KUKA KRL program: MyProgram_134().src

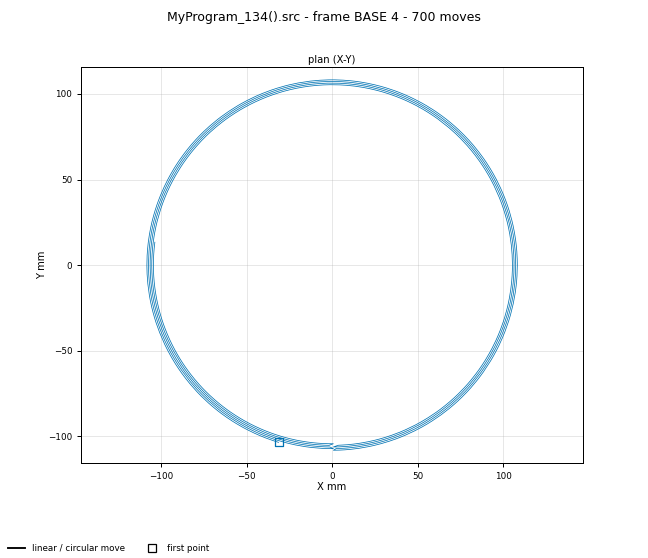
[picture p0: tool path of MyProgram_134().src in frame BASE 4, 700 of 700 moves have a stored position in this frame; points joined in program order, loops and branches not executed]
&ACCESS RVP
&REL 1
&PARAM TEMPLATE = C:\KRC\Roboter\Template\vorgabe
&PARAM EDITMASK = *
DEF MyProgram_134()
; ---- Setting reference (Base) ----
$BASE = BASE_DATA[4]

; --------------------------
; ---- Setting tool (TCP) ----
$TOOL = TOOL_DATA[3]
; --------------------------

$VEL.CP = VEL_APROX_PRINT
Startdeposition()
$VEL.CP = VEL_PRINT
LIN {X -31.2997,Y -103.6381,Z 109,A -111.208,B 24.951,C -1.6174,E1 24.9525,E2 197.031} C_DIS
LIN {X -34.6459,Y -102.5667,Z 109,A -112.942,B 24.9506,C -1.6238,E1 24.9479,E2 198.7528} C_DIS
LIN {X -39.0186,Y -100.9858,Z 109,A -115.4114,B 24.9505,C -1.6257,E1 24.9415,E2 201.2229} C_DIS
LIN {X -41.9877,Y -99.7862,Z 109,A -117.1477,B 24.9505,C -1.6258,E1 24.937,E2 202.9627} C_DIS
LIN {X -45.2763,Y -98.3388,Z 109,A -119.1694,B 24.9506,C -1.6232,E1 24.9318,E2 204.9956} C_DIS
LIN {X -49.3314,Y -96.3674,Z 109,A -121.2937,B 24.9498,C -1.6364,E1 24.9265,E2 207.094} C_DIS
LIN {X -51.851,Y -95.0358,Z 109,A -122.882,B 24.9498,C -1.6353,E1 24.9226,E2 208.6894} C_DIS
LIN {X -55.8456,Y -92.7447,Z 109,A -125.7501,B 24.9507,C -1.6221,E1 24.9156,E2 211.5976} C_DIS
LIN {X -58.5781,Y -91.0433,Z 109,A -127.0742,B 24.9496,C -1.6394,E1 24.9126,E2 212.8848} C_DIS
LIN {X -61.9141,Y -88.8083,Z 109,A -128.9557,B 24.9488,C -1.6523,E1 24.9083,E2 214.7419} C_DIS
LIN {X -64.9559,Y -86.6083,Z 109,A -130.8435,B 24.9484,C -1.6596,E1 24.9041,E2 216.6191} C_DIS
LIN {X -66.9949,Y -85.041,Z 109,A -133.1338,B 24.9504,C -1.6263,E1 24.8988,E2 218.9969} C_DIS
LIN {X -70.0734,Y -82.5228,Z 109,A -134.5366,B 24.9485,C -1.6572,E1 24.896,E2 220.3317} C_DIS
LIN {X -72.2415,Y -80.6314,Z 109,A -136.2176,B 24.9487,C -1.6541,E1 24.8924,E2 222.0266} C_DIS
LIN {X -76.5685,Y -76.5371,Z 109,A -139.3804,B 24.9483,C -1.6602,E1 24.8861,E2 225.188} C_DIS
LIN {X -78.8105,Y -74.2237,Z 109,A -141.1111,B 24.9482,C -1.663,E1 24.8827,E2 226.9196} C_DIS
LIN {X -82.7809,Y -69.7705,Z 109,A -144.1663,B 24.9475,C -1.6741,E1 24.8771,E2 229.9622} C_DIS
LIN {X -85.4607,Y -66.4602,Z 109,A -147.0858,B 24.9487,C -1.6544,E1 24.8719,E2 232.9421} C_DIS
LIN {X -87.8227,Y -63.3064,Z 109,A -148.5502,B 24.9469,C -1.6829,E1 24.8696,E2 234.3458} C_DIS
LIN {X -89.5892,Y -60.7786,Z 109,A -150.2841,B 24.9469,C -1.6832,E1 24.8669,E2 236.0876} C_DIS
LIN {X -91.4271,Y -57.9783,Z 109,A -152.4744,B 24.9476,C -1.6722,E1 24.8635,E2 238.3151} C_DIS
LIN {X -93.1735,Y -55.1267,Z 109,A -153.487,B 24.9455,C -1.7053,E1 24.8622,E2 239.2541} C_DIS
LIN {X -94.4849,Y -52.8476,Z 109,A -155.2178,B 24.9461,C -1.6963,E1 24.8597,E2 241.0155} C_DIS
LIN {X -96.0657,Y -49.9199,Z 109,A -157.1133,B 24.9461,C -1.6961,E1 24.8572,E2 242.9215} C_DIS
LIN {X -97.7535,Y -46.526,Z 109,A -158.9949,B 24.9454,C -1.7064,E1 24.8549,E2 244.7887} C_DIS
LIN {X -100.7843,Y -39.5322,Z 109,A -162.8386,B 24.9442,C -1.7251,E1 24.8508,E2 248.609} C_DIS
LIN {X -102.8692,Y -33.7398,Z 109,A -166.1714,B 24.9438,C -1.7319,E1 24.8476,E2 251.9445} C_DIS
LIN {X -103.7217,Y -31.018,Z 109,A -167.7303,B 24.9436,C -1.7347,E1 24.8463,E2 253.5058} C_DIS
LIN {X -104.5558,Y -28.0779,Z 109,A -169.4326,B 24.9435,C -1.7365,E1 24.8451,E2 255.2137} C_DIS
LIN {X -105.376,Y -24.8268,Z 109,A -171.3428,B 24.9435,C -1.7369,E1 24.8438,E2 257.134} C_DIS
LIN {X -106.1063,Y -21.4891,Z 109,A -173.1333,B 24.943,C -1.7432,E1 24.8427,E2 258.92} C_DIS
LIN {X -106.7849,Y -17.8116,Z 109,A -174.9667,B 24.9423,C -1.7548,E1 24.8419,E2 260.7366} C_DIS
LIN {X -107.7054,Y -10.9507,Z 109,A -178.2406,B 24.9406,C -1.7809,E1 24.8407,E2 263.968} C_DIS
LIN {X -108.1326,Y -5.2917,Z 109,A 177.367,B 24.9433,C -1.7395,E1 24.8399,E2 268.4854} C_DIS
LIN {X -108.26,Y -0.3831,Z 109,A 175.7447,B 24.9404,C -1.7835,E1 24.8398,E2 270.0125} C_DIS
LIN {X -108.1231,Y 5.4692,Z 109,A 171.9553,B 24.9414,C -1.7682,E1 24.8402,E2 273.8612} C_DIS
LIN {X -107.8794,Y 9.0831,Z 109,A 170.723,B 24.9393,C -1.7995,E1 24.8404,E2 275.0264} C_DIS
LIN {X -107.4684,Y 13.0778,Z 109,A 168.1987,B 24.9398,C -1.7917,E1 24.8412,E2 277.5844} C_DIS
LIN {X -106.7621,Y 17.9479,Z 109,A 165.7511,B 24.9389,C -1.8059,E1 24.8422,E2 280.0127} C_DIS
LIN {X -106.0692,Y 21.6699,Z 109,A 163.7287,B 24.9385,C -1.8116,E1 24.8433,E2 282.0333} C_DIS
LIN {X -105.3206,Y 25.064,Z 109,A 161.6321,B 24.9387,C -1.8081,E1 24.8446,E2 284.1507} C_DIS
LIN {X -104.4012,Y 28.6502,Z 109,A 159.8517,B 24.9379,C -1.8209,E1 24.8459,E2 285.911} C_DIS
LIN {X -103.4381,Y 31.9503,Z 109,A 158.0681,B 24.9374,C -1.8279,E1 24.8473,E2 287.688} C_DIS
LIN {X -102.395,Y 35.1552,Z 109,A 156.3651,B 24.9368,C -1.8365,E1 24.8488,E2 289.3805} C_DIS
LIN {X -101.522,Y 37.6008,Z 109,A 154.9641,B 24.9366,C -1.8398,E1 24.8501,E2 290.7815} C_DIS
LIN {X -100.3072,Y 40.7276,Z 109,A 153.1045,B 24.9364,C -1.8421,E1 24.852,E2 292.6458} C_DIS
LIN {X -98.0555,Y 45.8849,Z 109,A 150.153,B 24.9357,C -1.8522,E1 24.8554,E2 295.5897} C_DIS
LIN {X -95.9706,Y 50.1005,Z 109,A 147.8099,B 24.9348,C -1.865,E1 24.8583,E2 297.9148} C_DIS
LIN {X -94.6229,Y 52.6004,Z 109,A 146.1226,B 24.935,C -1.8626,E1 24.8606,E2 299.6168} C_DIS
LIN {X -92.3331,Y 56.5241,Z 109,A 143.8104,B 24.9342,C -1.8729,E1 24.8638,E2 301.9163} C_DIS
LIN {X -91.1364,Y 58.4331,Z 109,A 142.0785,B 24.9354,C -1.8564,E1 24.8665,E2 303.6963} C_DIS
LIN {X -89.2718,Y 61.2474,Z 109,A 140.5306,B 24.9344,C -1.8701,E1 24.8689,E2 305.2192} C_DIS
LIN {X -86.4338,Y 65.1882,Z 109,A 138.1976,B 24.9333,C -1.8859,E1 24.8727,E2 307.5257} C_DIS
LIN {X -84.5613,Y 67.6018,Z 109,A 136.5277,B 24.9332,C -1.8882,E1 24.8756,E2 309.198} C_DIS
LIN {X -82.1925,Y 70.4611,Z 109,A 134.7359,B 24.9323,C -1.8999,E1 24.8788,E2 310.9704} C_DIS
LIN {X -79.8747,Y 73.0774,Z 109,A 132.2119,B 24.9338,C -1.8795,E1 24.8836,E2 313.5543} C_DIS
LIN {X -77.5153,Y 75.578,Z 109,A 130.2995,B 24.9338,C -1.8805,E1 24.8873,E2 315.4724} C_DIS
LIN {X -74.9775,Y 78.0939,Z 109,A 128.917,B 24.932,C -1.9039,E1 24.89,E2 316.8048} C_DIS
LIN {X -71.5451,Y 81.2511,Z 109,A 126.0713,B 24.9326,C -1.8955,E1 24.896,E2 319.682} C_DIS
LIN {X -67.1017,Y 84.9566,Z 109,A 123.7193,B 24.9302,C -1.929,E1 24.9009,E2 321.9631} C_DIS
LIN {X -65.0027,Y 86.5731,Z 109,A 121.9258,B 24.9311,C -1.9172,E1 24.905,E2 323.7913} C_DIS
LIN {X -60.4243,Y 89.8291,Z 109,A 118.9522,B 24.9307,C -1.9231,E1 24.9118,E2 326.7609} C_DIS
LIN {X -55.121,Y 93.1769,Z 109,A 115.9848,B 24.9292,C -1.9427,E1 24.9187,E2 329.691} C_DIS
LIN {X -52.9651,Y 94.4192,Z 109,A 114.3034,B 24.9301,C -1.9312,E1 24.9228,E2 331.4049} C_DIS
LIN {X -49.4521,Y 96.3057,Z 109,A 111.2421,B 24.9324,C -1.8987,E1 24.9307,E2 334.5518} C_DIS
LIN {X -44.5516,Y 98.6682,Z 109,A 109.4911,B 24.929,C -1.946,E1 24.9348,E2 336.1947} C_DIS
LIN {X -40.7223,Y 100.3093,Z 109,A 106.7676,B 24.9302,C -1.9292,E1 24.9419,E2 338.9642} C_DIS
LIN {X -35.7507,Y 102.1869,Z 109,A 104.2114,B 24.9292,C -1.9427,E1 24.9486,E2 341.4935} C_DIS
LIN {X -32.0331,Y 103.4125,Z 109,A 102.2297,B 24.9288,C -1.9486,E1 24.9538,E2 343.4648} C_DIS
LIN {X -27.4862,Y 104.7142,Z 109,A 99.7876,B 24.9284,C -1.9536,E1 24.9604,E2 345.8989} C_DIS
LIN {X -25.0053,Y 105.3348,Z 109,A 97.4244,B 24.9312,C -1.9158,E1 24.9671,E2 348.355} C_DIS
LIN {X -19.867,Y 106.4234,Z 109,A 95.5962,B 24.9283,C -1.955,E1 24.9718,E2 350.0924} C_DIS
LIN {X -12.8383,Y 107.4965,Z 109,A 92.026,B 24.9276,C -1.965,E1 24.9816,E2 353.6416} C_DIS
LIN {X -7.2866,Y 108.0146,Z 109,A 88.6561,B 24.9287,C -1.9499,E1 24.9911,E2 357.0491} C_DIS
LIN {X -1.9168,Y 108.2432,Z 109,A 85.927,B 24.9283,C -1.9553,E1 24.9987,E2 359.7657} C_DIS
LIN {X 1.5277,Y 108.2504,Z 109,A 83.9851,B 24.9286,C -1.9509,E1 25.0041,E2 361.7179} C_DIS
LIN {X 6.494,Y 108.0662,Z 109,A 81.2757,B 24.9289,C -1.9479,E1 25.0117,E2 364.4337} C_DIS
LIN {X 10.3854,Y 107.7617,Z 109,A 79.4913,B 24.9281,C -1.9589,E1 25.0166,E2 366.1908} C_DIS
LIN {X 13.2983,Y 107.442,Z 109,A 77.4495,B 24.9295,C -1.939,E1 25.0224,E2 368.2785} C_DIS
LIN {X 16.5624,Y 106.9857,Z 109,A 76.1487,B 24.9282,C -1.9563,E1 25.0258,E2 369.5371} C_DIS
LIN {X 20.6241,Y 106.2776,Z 109,A 73.972,B 24.9282,C -1.9557,E1 25.0318,E2 371.7128} C_DIS
LIN {X 24.7533,Y 105.3922,Z 109,A 71.204,B 24.9299,C -1.933,E1 25.0395,E2 374.5307} C_DIS
LIN {X 28.4312,Y 104.4603,Z 109,A 69.5667,B 24.929,C -1.9467,E1 25.0438,E2 376.133} C_DIS
LIN {X 32.1117,Y 103.3881,Z 109,A 67.7029,B 24.9286,C -1.9519,E1 25.0487,E2 377.9812} C_DIS
LIN {X 36.1951,Y 102.0309,Z 109,A 65.4764,B 24.9286,C -1.9519,E1 25.0546,E2 380.203} C_DIS
LIN {X 39.034,Y 100.9799,Z 109,A 63.8342,B 24.9288,C -1.9488,E1 25.0589,E2 381.8493} C_DIS
LIN {X 42.0124,Y 99.7758,Z 109,A 62.1532,B 24.9288,C -1.9478,E1 25.0633,E2 383.5287} C_DIS
LIN {X 45.2347,Y 98.3581,Z 109,A 60.1584,B 24.9294,C -1.9402,E1 25.0684,E2 385.5365} C_DIS
LIN {X 48.122,Y 96.977,Z 109,A 58.5628,B 24.9293,C -1.9422,E1 25.0723,E2 387.1233} C_DIS
LIN {X 52.3281,Y 94.7735,Z 109,A 55.6623,B 24.9307,C -1.9228,E1 25.0796,E2 390.0613} C_DIS
LIN {X 55.2195,Y 93.1186,Z 109,A 54.3308,B 24.9296,C -1.9381,E1 25.0827,E2 391.3526} C_DIS
LIN {X 58.8637,Y 90.8599,Z 109,A 52.1495,B 24.9296,C -1.9382,E1 25.0878,E2 393.5266} C_DIS
LIN {X 60.952,Y 89.4718,Z 109,A 50.6676,B 24.9302,C -1.9296,E1 25.0913,E2 395.024} C_DIS
LIN {X 63.9983,Y 87.3183,Z 109,A 48.3971,B 24.9313,C -1.9138,E1 25.0965,E2 397.3238} C_DIS
LIN {X 66.611,Y 85.3444,Z 109,A 46.9917,B 24.9306,C -1.9243,E1 25.0995,E2 398.6993} C_DIS
LIN {X 69.1078,Y 83.3329,Z 109,A 45.361,B 24.9306,C -1.9239,E1 25.103,E2 400.3246} C_DIS
LIN {X 71.502,Y 81.2887,Z 109,A 43.5306,B 24.9313,C -1.9137,E1 25.1069,E2 402.172} C_DIS
LIN {X 74.3139,Y 78.7258,Z 109,A 41.6291,B 24.9313,C -1.9143,E1 25.1108,E2 404.0644} C_DIS
LIN {X 77.0481,Y 76.0516,Z 109,A 39.7051,B 24.9313,C -1.9143,E1 25.1146,E2 405.9804} C_DIS
LIN {X 80.2193,Y 72.7014,Z 109,A 37.1456,B 24.9321,C -1.9037,E1 25.1195,E2 408.5535} C_DIS
LIN {X 82.4514,Y 70.1572,Z 109,A 35.4807,B 24.932,C -1.905,E1 25.1225,E2 410.2079} C_DIS
LIN {X 84.4363,Y 67.7572,Z 109,A 33.8876,B 24.932,C -1.9034,E1 25.1253,E2 411.7973} C_DIS
LIN {X 85.8314,Y 65.979,Z 109,A 32.5901,B 24.9326,C -1.8962,E1 25.1276,E2 413.1058} C_DIS
LIN {X 88.5381,Y 62.3028,Z 109,A 30.3143,B 24.9326,C -1.8961,E1 25.1313,E2 415.3708} C_DIS
LIN {X 90.0935,Y 60.0307,Z 109,A 28.5381,B 24.9338,C -1.8787,E1 25.1341,E2 417.1793} C_DIS
LIN {X 92.5262,Y 56.2063,Z 109,A 26.4178,B 24.9334,C -1.8843,E1 25.1372,E2 419.2755} C_DIS
LIN {X 94.3098,Y 53.1611,Z 109,A 24.4436,B 24.9341,C -1.8747,E1 25.14,E2 421.2622} C_DIS
LIN {X 96.0099,Y 50.0258,Z 109,A 22.33,B 24.9352,C -1.8597,E1 25.1428,E2 423.3999} C_DIS
LIN {X 98.5399,Y 44.8363,Z 109,A 19.2343,B 24.9359,C -1.8493,E1 25.1464,E2 426.5035} C_DIS
LIN {X 100.374,Y 40.5635,Z 109,A 17.2053,B 24.9351,C -1.8608,E1 25.1486,E2 428.4943} C_DIS
LIN {X 101.4884,Y 37.6928,Z 109,A 15.5397,B 24.9355,C -1.8544,E1 25.1502,E2 430.1657} C_DIS
LIN {X 102.5248,Y 34.7701,Z 109,A 13.9067,B 24.9359,C -1.8499,E1 25.1517,E2 431.8002} C_DIS
LIN {X 103.6373,Y 31.3027,Z 109,A 11.0696,B 24.9389,C -1.8048,E1 25.1541,E2 434.7274} C_DIS
LIN {X 105.0923,Y 25.9998,Z 109,A 9.2285,B 24.9364,C -1.842,E1 25.1553,E2 436.4702} C_DIS
LIN {X 105.7766,Y 23.056,Z 109,A 6.8963,B 24.9389,C -1.8052,E1 25.1568,E2 438.8755} C_DIS
LIN {X 106.6045,Y 18.8636,Z 109,A 5.3215,B 24.9374,C -1.8279,E1 25.1575,E2 440.3877} C_DIS
LIN {X 107.307,Y 14.3408,Z 109,A 2.8574,B 24.938,C -1.8184,E1 25.1585,E2 442.8597} C_DIS
LIN {X 107.6715,Y 11.2741,Z 109,A 1.2544,B 24.9383,C -1.8145,E1 25.159,E2 444.4623} C_DIS
LIN {X 107.9616,Y 8.0544,Z 109,A -0.6416,B 24.9392,C -1.8009,E1 25.1595,E2 446.3792} C_DIS
LIN {X 108.2051,Y 3.4543,Z 109,A -2.8585,B 24.9391,C -1.8027,E1 25.1597,E2 448.5787} C_DIS
LIN {X 108.2615,Y -0.0902,Z 109,A -5.0651,B 24.9405,C -1.7822,E1 25.1597,E2 450.8205} C_DIS
LIN {X 108.0695,Y -6.4382,Z 109,A -7.9587,B 24.9398,C -1.7917,E1 25.1595,E2 453.6744} C_DIS
LIN {X 107.9045,Y -8.769,Z 109,A -9.2762,B 24.9403,C -1.7842,E1 25.1592,E2 455.0019} C_DIS
LIN {X 107.5873,Y -12.0626,Z 109,A -11.5818,B 24.9423,C -1.7543,E1 25.1585,E2 457.3643} C_DIS
LIN {X 107.0812,Y -15.9445,Z 109,A -13.1939,B 24.9414,C -1.7676,E1 25.1578,E2 458.9355} C_DIS
LIN {X 105.9091,Y -22.4482,Z 109,A -16.4849,B 24.9416,C -1.7653,E1 25.1562,E2 462.2126} C_DIS
LIN {X 104.2843,Y -29.0728,Z 109,A -20.3507,B 24.9431,C -1.7426,E1 25.1535,E2 466.1097} C_DIS
LIN {X 103.207,Y -32.6958,Z 109,A -22.293,B 24.9433,C -1.7388,E1 25.1519,E2 468.0499} C_DIS
LIN {X 100.9919,Y -39.0036,Z 109,A -25.5638,B 24.9433,C -1.7394,E1 25.1488,E2 471.3009} C_DIS
LIN {X 99.6017,Y -42.4255,Z 109,A -27.6708,B 24.9441,C -1.7268,E1 25.1465,E2 473.4262} C_DIS
LIN {X 97.647,Y -46.7477,Z 109,A -30.0763,B 24.9443,C -1.7237,E1 25.1437,E2 475.8258} C_DIS
LIN {X 96.2159,Y -49.6277,Z 109,A -32.3155,B 24.9461,C -1.6953,E1 25.1408,E2 478.1201} C_DIS
LIN {X 94.4054,Y -52.9898,Z 109,A -34.039,B 24.9457,C -1.7023,E1 25.1385,E2 479.8183} C_DIS
LIN {X 92.7773,Y -55.7932,Z 109,A -35.5303,B 24.9454,C -1.707,E1 25.1364,E2 481.2909} C_DIS
LIN {X 88.4025,Y -62.4938,Z 109,A -39.5442,B 24.9455,C -1.7046,E1 25.1302,E2 485.2903} C_DIS
LIN {X 86.659,Y -64.8884,Z 109,A -41.6504,B 24.9473,C -1.677,E1 25.1266,E2 487.4516} C_DIS
LIN {X 84.6487,Y -67.4912,Z 109,A -42.9071,B 24.9463,C -1.6932,E1 25.1245,E2 488.6641} C_DIS
LIN {X 81.0925,Y -71.7264,Z 109,A -46.0205,B 24.9473,C -1.6775,E1 25.1189,E2 491.8005} C_DIS
LIN {X 78.4842,Y -74.5708,Z 109,A -48.4719,B 24.9487,C -1.6548,E1 25.1141,E2 494.2948} C_DIS
LIN {X 75.8147,Y -77.2821,Z 109,A -50.4406,B 24.9489,C -1.6518,E1 25.1102,E2 496.2623} C_DIS
LIN {X 73.153,Y -79.8053,Z 109,A -51.4554,B 24.9467,C -1.687,E1 25.1083,E2 497.1898} C_DIS
LIN {X 71.307,Y -81.4591,Z 109,A -53.2526,B 24.9482,C -1.663,E1 25.1044,E2 499.0365} C_DIS
LIN {X 68.2255,Y -84.0568,Z 109,A -55.3008,B 24.9482,C -1.6619,E1 25.1,E2 501.0796} C_DIS
LIN {X 63.7057,Y -87.5325,Z 109,A -58.1189,B 24.9482,C -1.6639,E1 25.0938,E2 503.8825} C_DIS
LIN {X 58.6126,Y -91.0211,Z 109,A -61.9488,B 24.95,C -1.6334,E1 25.0848,E2 507.7717} C_DIS
LIN {X 55.7926,Y -92.7777,Z 109,A -63.4928,B 24.9497,C -1.6392,E1 25.0811,E2 509.2973} C_DIS
LIN {X 52.2469,Y -94.8203,Z 109,A -66.155,B 24.9512,C -1.6144,E1 25.0745,E2 512.0102} C_DIS
LIN {X 48.3312,Y -96.8733,Z 109,A -67.5412,B 24.9489,C -1.6507,E1 25.0713,E2 513.3068} C_DIS
LIN {X 42.9618,Y -99.3712,Z 109,A -70.8479,B 24.9497,C -1.6384,E1 25.0629,E2 516.6342} C_DIS
LIN {X 39.8739,Y -100.65,Z 109,A -72.682,B 24.95,C -1.6331,E1 25.0581,E2 518.4766} C_DIS
LIN {X 37.1385,Y -101.6907,Z 109,A -74.5311,B 24.9509,C -1.6185,E1 25.0532,E2 520.3565} C_DIS
LIN {X 33.4075,Y -102.9767,Z 109,A -76.3201,B 24.9503,C -1.6284,E1 25.0485,E2 522.1185} C_DIS
LIN {X 28.7106,Y -104.3849,Z 109,A -79.2516,B 24.9513,C -1.6115,E1 25.0405,E2 525.0851} C_DIS
LIN {X 24.3052,Y -105.4965,Z 109,A -81.2451,B 24.9504,C -1.6262,E1 25.0352,E2 527.041} C_DIS
LIN {X 21.6093,Y -106.0817,Z 109,A -82.7145,B 24.9506,C -1.6245,E1 25.0312,E2 528.5125} C_DIS
LIN {X 15.8857,Y -107.0903,Z 109,A -85.9029,B 24.951,C -1.6174,E1 25.0224,E2 531.7143} C_DIS
LIN {X 10.6167,Y -107.7403,Z 109,A -88.5635,B 24.9507,C -1.6219,E1 25.015,E2 534.3625} C_DIS
LIN {X 7.4584,Y -108.003,Z 109,A -90.2773,B 24.9508,C -1.6196,E1 25.0102,E2 536.0808} C_DIS
LIN {X 4.5496,Y -108.1645,Z 109,A -92.1603,B 24.9517,C -1.6051,E1 25.0049,E2 537.9977} C_DIS
LIN {X 0.7592,Y -108.2524,Z 109,A -93.6271,B 24.9504,C -1.6266,E1 25.001,E2 539.4131} C_DIS
Enddeposition()
LIN {X 0.7592,Y -108.2524,Z 109,A -93.6271,B 24.9504,C -1.6266,E1 25.001,E2 539.4131} C_DIS
Startdeposition()
$VEL.CP = VEL_PRINT
LIN {X 2.4015,Y -107.2831,Z 109,A -92.1371,B 24.9478,C -1.6685,E1 25.0054,E2 537.8241} C_DIS
LIN {X 7.3,Y -107.0605,Z 109,A -89.6064,B 24.948,C -1.666,E1 25.0124,E2 535.3003} C_DIS
LIN {X 9.9244,Y -106.8492,Z 109,A -87.3231,B 24.9456,C -1.7033,E1 25.019,E2 532.93} C_DIS
LIN {X 15.1446,Y -106.2351,Z 109,A -85.7505,B 24.9488,C -1.6537,E1 25.023,E2 531.4762} C_DIS
LIN {X 22.3374,Y -104.9599,Z 109,A -80.7234,B 24.9456,C -1.7039,E1 25.0371,E2 526.336} C_DIS
LIN {X 27.0253,Y -103.8508,Z 109,A -78.2009,B 24.9456,C -1.7045,E1 25.0439,E2 523.816} C_DIS
LIN {X 31.5174,Y -102.5767,Z 109,A -76.4123,B 24.9473,C -1.6775,E1 25.0486,E2 522.0943} C_DIS
LIN {X 35.062,Y -101.4206,Z 109,A -73.8334,B 24.9455,C -1.705,E1 25.0555,E2 519.4556} C_DIS
LIN {X 39.0029,Y -99.9704,Z 109,A -72.2135,B 24.947,C -1.6816,E1 25.0596,E2 517.8944} C_DIS
LIN {X 42.1902,Y -98.6689,Z 109,A -70.0802,B 24.946,C -1.6968,E1 25.0652,E2 515.7302} C_DIS
LIN {X 48.3594,Y -95.7962,Z 109,A -66.2547,B 24.9451,C -1.7109,E1 25.0748,E2 511.8815} C_DIS
LIN {X 51.7439,Y -94.0119,Z 109,A -64.6591,B 24.9461,C -1.6953,E1 25.0786,E2 510.3273} C_DIS
LIN {X 54.0662,Y -92.6956,Z 109,A -63.1494,B 24.9457,C -1.7015,E1 25.0823,E2 508.8075} C_DIS
LIN {X 57.8716,Y -90.3666,Z 109,A -60.4791,B 24.9447,C -1.7186,E1 25.0887,E2 506.1055} C_DIS
LIN {X 60.8527,Y -88.3868,Z 109,A -58.8734,B 24.9452,C -1.7093,E1 25.0923,E2 504.5273} C_DIS
LIN {X 64.0094,Y -86.1299,Z 109,A -56.3789,B 24.9438,C -1.7319,E1 25.098,E2 501.9883} C_DIS
LIN {X 67.2506,Y -83.6228,Z 109,A -54.3668,B 24.944,C -1.7291,E1 25.1024,E2 499.9903} C_DIS
LIN {X 69.9036,Y -81.418,Z 109,A -52.8071,B 24.9445,C -1.721,E1 25.1056,E2 498.4557} C_DIS
LIN {X 73.9766,Y -77.7342,Z 109,A -49.8866,B 24.9441,C -1.7275,E1 25.1116,E2 495.5319} C_DIS
LIN {X 77.6008,Y -74.1172,Z 109,A -46.8866,B 24.9429,C -1.7458,E1 25.1175,E2 492.5015} C_DIS
LIN {X 79.9717,Y -71.5526,Z 109,A -45.7902,B 24.9447,C -1.7172,E1 25.1195,E2 491.4775} C_DIS
LIN {X 82.2811,Y -68.8856,Z 109,A -43.4335,B 24.9431,C -1.7426,E1 25.1238,E2 489.0715} C_DIS
LIN {X 86.512,Y -63.4897,Z 109,A -39.9572,B 24.943,C -1.7444,E1 25.1297,E2 485.6074} C_DIS
LIN {X 88.6784,Y -60.4275,Z 109,A -37.3619,B 24.9409,C -1.776,E1 25.1339,E2 482.9503} C_DIS
LIN {X 90.951,Y -56.9488,Z 109,A -35.817,B 24.9424,C -1.7528,E1 25.1361,E2 481.4681} C_DIS
LIN {X 93.5825,Y -52.513,Z 109,A -33.3223,B 24.9426,C -1.7494,E1 25.1396,E2 478.9941} C_DIS
LIN {X 95.638,Y -48.6688,Z 109,A -30.8531,B 24.9418,C -1.7625,E1 25.1429,E2 476.5071} C_DIS
LIN {X 98.0003,Y -43.7187,Z 109,A -27.7554,B 24.9407,C -1.7787,E1 25.1466,E2 473.3877} C_DIS
LIN {X 99.2942,Y -40.6937,Z 109,A -24.7809,B 24.9367,C -1.8382,E1 25.1498,E2 470.2894} C_DIS
LIN {X 101.7194,Y -34.1821,Z 109,A -22.3793,B 24.9398,C -1.7917,E1 25.1519,E2 468.0111} C_DIS
LIN {X 103.0224,Y -30.0314,Z 109,A -18.8715,B 24.9357,C -1.8516,E1 25.1548,E2 464.3819} C_DIS
LIN {X 104.6773,Y -23.6262,Z 109,A -16.5498,B 24.9387,C -1.8091,E1 25.1562,E2 462.1741} C_DIS
LIN {X 105.8865,Y -17.4179,Z 109,A -13.3657,B 24.9385,C -1.8114,E1 25.1578,E2 459.0029} C_DIS
LIN {X 106.7959,Y -10.5021,Z 109,A -9.5749,B 24.9375,C -1.8263,E1 25.1591,E2 455.1994} C_DIS
LIN {X 107.1239,Y -6.3146,Z 109,A -7.0784,B 24.9362,C -1.8448,E1 25.1596,E2 452.6742} C_DIS
LIN {X 107.3109,Y -0.0133,Z 109,A -3.7996,B 24.9357,C -1.8518,E1 25.1598,E2 449.3983} C_DIS
LIN {X 107.1459,Y 5.9166,Z 109,A -0.382,B 24.9342,C -1.8731,E1 25.1594,E2 445.9508} C_DIS
LIN {X 106.9036,Y 9.3357,Z 109,A 1.1087,B 24.9349,C -1.864,E1 25.159,E2 444.4904} C_DIS
LIN {X 106.4672,Y 13.4209,Z 109,A 3.9297,B 24.9324,C -1.8987,E1 25.1581,E2 441.6043} C_DIS
LIN {X 105.7868,Y 18.0138,Z 109,A 5.6559,B 24.9342,C -1.8733,E1 25.1573,E2 439.9481} C_DIS
LIN {X 104.7408,Y 23.3421,Z 109,A 8.6501,B 24.9333,C -1.8865,E1 25.1556,E2 436.9401} C_DIS
LIN {X 102.8364,Y 30.6585,Z 109,A 12.6137,B 24.9326,C -1.8957,E1 25.1527,E2 432.9778} C_DIS
LIN {X 101.7031,Y 34.2305,Z 109,A 14.4752,B 24.9326,C -1.8957,E1 25.1511,E2 431.1269} C_DIS
LIN {X 100.9298,Y 36.449,Z 109,A 15.9956,B 24.9315,C -1.911,E1 25.1497,E2 429.5788} C_DIS
LIN {X 99.4457,Y 40.3215,Z 109,A 17.7528,B 24.9325,C -1.8976,E1 25.1479,E2 427.863} C_DIS
LIN {X 97.5132,Y 44.7958,Z 109,A 20.4267,B 24.9317,C -1.9082,E1 25.1449,E2 425.1788} C_DIS
LIN {X 95.2524,Y 49.4233,Z 109,A 23.4417,B 24.9304,C -1.9273,E1 25.1411,E2 422.1346} C_DIS
LIN {X 93.9139,Y 51.9195,Z 109,A 24.8609,B 24.9304,C -1.9274,E1 25.1392,E2 420.7226} C_DIS
LIN {X 92.2424,Y 54.8329,Z 109,A 26.5534,B 24.9304,C -1.9279,E1 25.1369,E2 419.0376} C_DIS
LIN {X 90.7027,Y 57.3463,Z 109,A 28.5934,B 24.9285,C -1.9522,E1 25.1338,E2 416.9507} C_DIS
LIN {X 88.8829,Y 60.1255,Z 109,A 29.5508,B 24.9308,C -1.9216,E1 25.1324,E2 416.0702} C_DIS
LIN {X 86.4079,Y 63.6318,Z 109,A 32.3086,B 24.9289,C -1.9474,E1 25.1279,E2 413.265} C_DIS
LIN {X 84.1958,Y 66.5305,Z 109,A 34.2522,B 24.9286,C -1.9519,E1 25.1245,E2 411.3198} C_DIS
LIN {X 81.8561,Y 69.3895,Z 109,A 36.0807,B 24.9286,C -1.9504,E1 25.1213,E2 409.5034} C_DIS
LIN {X 80.1087,Y 71.3996,Z 109,A 38.2235,B 24.9262,C -1.9846,E1 25.1171,E2 407.2892} C_DIS
LIN {X 76.9995,Y 74.7426,Z 109,A 40.0165,B 24.9278,C -1.9623,E1 25.1138,E2 405.5568} C_DIS
LIN {X 74.5542,Y 77.1812,Z 109,A 41.7828,B 24.9278,C -1.9629,E1 25.1103,E2 403.7965} C_DIS
LIN {X 72.5161,Y 79.0991,Z 109,A 43.591,B 24.9265,C -1.9793,E1 25.1065,E2 401.9567} C_DIS
LIN {X 68.7614,Y 82.3843,Z 109,A 45.917,B 24.9272,C -1.9702,E1 25.1016,E2 399.6614} C_DIS
LIN {X 63.3051,Y 86.6471,Z 109,A 49.6005,B 24.9268,C -1.9762,E1 25.0935,E2 395.9771} C_DIS
LIN {X 59.3516,Y 89.4022,Z 109,A 51.9347,B 24.9272,C -1.9705,E1 25.0882,E2 393.6644} C_DIS
LIN {X 56.1222,Y 91.4645,Z 109,A 54.3126,B 24.9259,C -1.9875,E1 25.0825,E2 391.2538} C_DIS
LIN {X 50.5379,Y 94.6654,Z 109,A 57.7267,B 24.9256,C -1.9914,E1 25.0741,E2 387.8406} C_DIS
LIN {X 47.3874,Y 96.2797,Z 109,A 59.5888,B 24.9256,C -1.9927,E1 25.0695,E2 385.9806} C_DIS
LIN {X 43.6461,Y 98.0332,Z 109,A 61.7415,B 24.9256,C -1.993,E1 25.064,E2 383.8326} C_DIS
LIN {X 40.6782,Y 99.3005,Z 109,A 63.4056,B 24.9256,C -1.9924,E1 25.0598,E2 382.1737} C_DIS
LIN {X 37.5044,Y 100.5433,Z 109,A 65.0802,B 24.9259,C -1.9882,E1 25.0554,E2 380.5128} C_DIS
LIN {X 33.51,Y 101.944,Z 109,A 67.5078,B 24.9252,C -1.997,E1 25.049,E2 378.0691} C_DIS
LIN {X 30.5096,Y 102.8806,Z 109,A 69.1805,B 24.9252,C -1.9981,E1 25.0445,E2 376.3969} C_DIS
LIN {X 23.2494,Y 104.761,Z 109,A 73.2483,B 24.9248,C -2.0029,E1 25.0335,E2 372.3235} C_DIS
LIN {X 20.4076,Y 105.3508,Z 109,A 75.2324,B 24.9234,C -2.0213,E1 25.0279,E2 370.2982} C_DIS
LIN {X 16.7514,Y 105.9942,Z 109,A 76.4916,B 24.9256,C -1.9926,E1 25.0247,E2 369.1083} C_DIS
LIN {X 11.9085,Y 106.6479,Z 109,A 79.3813,B 24.9247,C -2.0044,E1 25.0166,E2 366.1929} C_DIS
LIN {X 9.3586,Y 106.9014,Z 109,A 81.2199,B 24.9232,C -2.0236,E1 25.0113,E2 364.3099} C_DIS
LIN {X 5.6035,Y 107.1632,Z 109,A 82.7189,B 24.9248,C -2.0029,E1 25.0073,E2 362.8605} C_DIS
LIN {X 1.4493,Y 107.3006,Z 109,A 85.0483,B 24.9245,C -2.0071,E1 25.0008,E2 360.5216} C_DIS
LIN {X -1.6403,Y 107.2971,Z 109,A 87.2873,B 24.9227,C -2.0303,E1 24.9944,E2 358.2273} C_DIS
LIN {X -6.1999,Y 107.1302,Z 109,A 88.7869,B 24.9256,C -1.992,E1 24.9904,E2 356.8183} C_DIS
LIN {X -9.791,Y 106.8615,Z 109,A 91.1853,B 24.9242,C -2.01,E1 24.9836,E2 354.3761} C_DIS
LIN {X -13.1488,Y 106.5024,Z 109,A 93.7976,B 24.9219,C -2.0412,E1 24.9762,E2 351.6879} C_DIS
LIN {X -18.9818,Y 105.6169,Z 109,A 95.502,B 24.9264,C -1.9816,E1 24.9719,E2 350.1234} C_DIS
LIN {X -24.3959,Y 104.4995,Z 109,A 98.9665,B 24.9251,C -1.999,E1 24.9623,E2 346.6133} C_DIS
LIN {X -27.8489,Y 103.6325,Z 109,A 101.1871,B 24.9243,C -2.0096,E1 24.9562,E2 344.3641} C_DIS
LIN {X -31.2039,Y 102.6739,Z 109,A 102.7969,B 24.9252,C -1.9976,E1 24.952,E2 342.7802} C_DIS
LIN {X -35.1778,Y 101.38,Z 109,A 104.6462,B 24.9265,C -1.9801,E1 24.9472,E2 340.9691} C_DIS
LIN {X -42.2774,Y 98.6321,Z 109,A 109.0464,B 24.9259,C -1.9874,E1 24.9357,E2 336.542} C_DIS
LIN {X -45.475,Y 97.1973,Z 109,A 110.7216,B 24.9267,C -1.977,E1 24.9315,E2 334.8874} C_DIS
LIN {X -48.8786,Y 95.5308,Z 109,A 113.2545,B 24.9255,C -1.9933,E1 24.9251,E2 332.309} C_DIS
LIN {X -51.8578,Y 93.9484,Z 109,A 114.7159,B 24.9267,C -1.9771,E1 24.9216,E2 330.8819} C_DIS
LIN {X -54.3636,Y 92.5198,Z 109,A 116.9238,B 24.925,C -2,E1 24.9161,E2 328.6128} C_DIS
LIN {X -58.2672,Y 90.1126,Z 109,A 118.6017,B 24.9275,C -1.9658,E1 24.9123,E2 327.0111} C_DIS
LIN {X -62.8626,Y 86.9711,Z 109,A 121.7086,B 24.9276,C -1.9649,E1 24.9052,E2 323.8957} C_DIS
LIN {X -64.9453,Y 85.4268,Z 109,A 123.3527,B 24.9271,C -1.9718,E1 24.9015,E2 322.2291} C_DIS
LIN {X -68.5158,Y 82.5883,Z 109,A 125.4938,B 24.9283,C -1.9553,E1 24.8969,E2 320.1192} C_DIS
LIN {X -72.8818,Y 78.7635,Z 109,A 128.5366,B 24.929,C -1.946,E1 24.8906,E2 317.0864} C_DIS
LIN {X -75.2388,Y 76.5142,Z 109,A 130.4655,B 24.9288,C -1.949,E1 24.8867,E2 315.1424} C_DIS
LIN {X -78.3274,Y 73.3493,Z 109,A 133.2695,B 24.928,C -1.9599,E1 24.8812,E2 312.3004} C_DIS
LIN {X -80.9104,Y 70.4895,Z 109,A 134.7322,B 24.93,C -1.9322,E1 24.8786,E2 310.897} C_DIS
LIN {X -83.8322,Y 66.9906,Z 109,A 137.2974,B 24.9301,C -1.9307,E1 24.8741,E2 308.3235} C_DIS
LIN {X -87.4418,Y 62.2029,Z 109,A 140.4606,B 24.9308,C -1.9206,E1 24.8688,E2 305.1692} C_DIS
LIN {X -90.393,Y 57.8305,Z 109,A 143.1872,B 24.9317,C -1.9093,E1 24.8646,E2 302.4558} C_DIS
LIN {X -92.6513,Y 54.1411,Z 109,A 145.7987,B 24.9313,C -1.9139,E1 24.8609,E2 299.82} C_DIS
LIN {X -94.7018,Y 50.4686,Z 109,A 148.2128,B 24.9313,C -1.9135,E1 24.8576,E2 297.394} C_DIS
LIN {X -96.9447,Y 46.0128,Z 109,A 151.2091,B 24.931,C -1.918,E1 24.854,E2 294.3708} C_DIS
LIN {X -98.7027,Y 42.1099,Z 109,A 152.9035,B 24.9331,C -1.889,E1 24.8522,E2 292.7362} C_DIS
LIN {X -99.9741,Y 38.9936,Z 109,A 154.7093,B 24.9335,C -1.8838,E1 24.8503,E2 290.9327} C_DIS
LIN {X -101.2843,Y 35.4506,Z 109,A 156.6996,B 24.934,C -1.8765,E1 24.8484,E2 288.9484} C_DIS
LIN {X -102.4242,Y 32.0092,Z 109,A 158.6774,B 24.9343,C -1.872,E1 24.8467,E2 286.9701} C_DIS
LIN {X -103.3265,Y 28.9649,Z 109,A 160.8429,B 24.9335,C -1.8841,E1 24.845,E2 284.7632} C_DIS
LIN {X -104.2366,Y 25.4949,Z 109,A 162.2844,B 24.9351,C -1.8604,E1 24.8441,E2 283.3698} C_DIS
LIN {X -105.0226,Y 22.039,Z 109,A 164.2247,B 24.9354,C -1.8561,E1 24.8429,E2 281.4283} C_DIS
LIN {X -105.6398,Y 18.8545,Z 109,A 165.8351,B 24.9361,C -1.8461,E1 24.8421,E2 279.8324} C_DIS
LIN {X -106.3594,Y 14.2529,Z 109,A 168.4862,B 24.9363,C -1.8441,E1 24.841,E2 277.1702} C_DIS
LIN {X -106.7749,Y 10.7048,Z 109,A 170.4375,B 24.9366,C -1.8395,E1 24.8404,E2 275.2181} C_DIS
LIN {X -107.0138,Y 7.9767,Z 109,A 172.0983,B 24.9364,C -1.8421,E1 24.8401,E2 273.5411} C_DIS
LIN {X -107.3016,Y 1.3973,Z 109,A 175.4547,B 24.9376,C -1.8248,E1 24.8398,E2 270.2058} C_DIS
LIN {X -107.2935,Y -1.835,Z 109,A 177.6229,B 24.9368,C -1.8356,E1 24.8398,E2 267.9987} C_DIS
LIN {X -107.1651,Y -5.5692,Z 109,A 179.7464,B 24.937,C -1.834,E1 24.8402,E2 265.8662} C_DIS
LIN {X -106.8691,Y -9.709,Z 109,A -178.6495,B 24.939,C -1.8042,E1 24.8406,E2 264.3238} C_DIS
LIN {X -106.0694,Y -16.2652,Z 109,A -174.992,B 24.9394,C -1.7978,E1 24.8419,E2 260.6597} C_DIS
LIN {X -105.3756,Y -20.2787,Z 109,A -172.9188,B 24.9401,C -1.7872,E1 24.8429,E2 258.5994} C_DIS
LIN {X -104.6684,Y -23.6648,Z 109,A -171.0599,B 24.9405,C -1.7818,E1 24.844,E2 256.7423} C_DIS
LIN {X -103.9287,Y -26.7223,Z 109,A -169.376,B 24.9408,C -1.7768,E1 24.8452,E2 255.0605} C_DIS
LIN {X -102.9513,Y -30.2713,Z 109,A -167.2785,B 24.9408,C -1.7757,E1 24.8468,E2 252.9535} C_DIS
LIN {X -102.0017,Y -33.3315,Z 109,A -165.0765,B 24.94,C -1.789,E1 24.8487,E2 250.7072} C_DIS
LIN {X -100.698,Y -37.0838,Z 109,A -163.4218,B 24.9416,C -1.7652,E1 24.8503,E2 249.1} C_DIS
LIN {X -99.6798,Y -39.7426,Z 109,A -161.1098,B 24.9399,C -1.7906,E1 24.8528,E2 246.7144} C_DIS
LIN {X -97.6352,Y -44.5293,Z 109,A -159.0677,B 24.9423,C -1.7547,E1 24.855,E2 244.7466} C_DIS
LIN {X -96.171,Y -47.6066,Z 109,A -157.3283,B 24.9428,C -1.7466,E1 24.8571,E2 243.0172} C_DIS
LIN {X -94.2825,Y -51.2451,Z 109,A -155.1512,B 24.9432,C -1.7402,E1 24.8599,E2 240.8439} C_DIS
LIN {X -92.5148,Y -54.3722,Z 109,A -153.0656,B 24.9432,C -1.7413,E1 24.8629,E2 238.7447} C_DIS
LIN {X -89.8609,Y -58.6558,Z 109,A -150.4735,B 24.9439,C -1.7305,E1 24.8667,E2 236.1652} C_DIS
LIN {X -88.0065,Y -61.4014,Z 109,A -148.7442,B 24.9443,C -1.7246,E1 24.8695,E2 234.4416} C_DIS
LIN {X -82.9104,Y -68.1282,Z 109,A -143.0726,B 24.942,C -1.7584,E1 24.8795,E2 228.6625} C_DIS
LIN {X -78.792,Y -72.8508,Z 109,A -140.7284,B 24.9451,C -1.7122,E1 24.8837,E2 226.418} C_DIS
LIN {X -76.3285,Y -75.4268,Z 109,A -137.8403,B 24.9428,C -1.7463,E1 24.8896,E2 223.4364} C_DIS
LIN {X -71.8815,Y -79.6772,Z 109,A -135.6344,B 24.946,C -1.6977,E1 24.8938,E2 221.3374} C_DIS
LIN {X -66.1336,Y -84.5095,Z 109,A -131.4857,B 24.9461,C -1.6954,E1 24.9028,E2 217.1783} C_DIS
LIN {X -63.9353,Y -86.1855,Z 109,A -129.7662,B 24.9457,C -1.7023,E1 24.9067,E2 215.4363} C_DIS
LIN {X -59.355,Y -89.3999,Z 109,A -127.1069,B 24.9468,C -1.6846,E1 24.9128,E2 212.8102} C_DIS
LIN {X -53.7857,Y -92.8573,Z 109,A -123.5948,B 24.9471,C -1.6798,E1 24.9211,E2 209.2986} C_DIS
LIN {X -50.6766,Y -94.5909,Z 109,A -121.5964,B 24.9471,C -1.681,E1 24.926,E2 207.2916} C_DIS
LIN {X -47.6393,Y -96.1548,Z 109,A -119.9067,B 24.9475,C -1.6735,E1 24.9302,E2 205.6153} C_DIS
LIN {X -44.5558,Y -97.6232,Z 109,A -117.962,B 24.9474,C -1.6761,E1 24.9352,E2 203.6594} C_DIS
LIN {X -41.2211,Y -99.0773,Z 109,A -116.1862,B 24.9479,C -1.6675,E1 24.9397,E2 201.9} C_DIS
LIN {X -36.1456,Y -101.0404,Z 109,A -113.1368,B 24.9477,C -1.6705,E1 24.9477,E2 198.8372} C_DIS
LIN {X -33.099,Y -102.077,Z 109,A -111.4842,B 24.948,C -1.6665,E1 24.9521,E2 197.191} C_DIS
LIN {X -26.1434,Y -104.0775,Z 109,A -107.5151,B 24.9479,C -1.6681,E1 24.9628,E2 193.2118} C_DIS
LIN {X -21.5399,Y -105.1251,Z 109,A -104.9757,B 24.9479,C -1.6677,E1 24.9697,E2 190.6702} C_DIS
LIN {X -15.9156,Y -106.1234,Z 109,A -101.9919,B 24.9481,C -1.6641,E1 24.9779,E2 187.6923} C_DIS
LIN {X -12.0149,Y -106.6354,Z 109,A -99.5383,B 24.9472,C -1.6781,E1 24.9848,E2 185.2037} C_DIS
LIN {X -5.7091,Y -107.1574,Z 109,A -96.5066,B 24.9481,C -1.6639,E1 24.9932,E2 182.2044} C_DIS
LIN {X -2.1546,Y -107.2876,Z 109,A -94.7932,B 24.9486,C -1.6566,E1 24.9979,E2 180.5081} C_DIS
LIN {X 0.7531,Y -107.2936,Z 109,A -93.5307,B 24.9493,C -1.6453,E1 25.0014,E2 179.2724} C_DIS
Enddeposition()
LIN {X 0.7531,Y -107.2936,Z 109,A -93.5307,B 24.9493,C -1.6453,E1 25.0014,E2 179.2724} C_DIS
Startdeposition()
$VEL.CP = VEL_PRINT
LIN {X -1.3601,Y -106.3511,Z 109,A -94.9609,B 24.949,C -1.6497,E1 24.9974,E2 180.6922} C_DIS
LIN {X -3.9218,Y -106.2876,Z 109,A -97.1151,B 24.9509,C -1.6189,E1 24.9912,E2 182.9199} C_DIS
LIN {X -8.1816,Y -106.0433,Z 109,A -99.3995,B 24.9509,C -1.6195,E1 24.9848,E2 185.2037} C_DIS
LIN {X -12.4229,Y -105.6301,Z 109,A -101.046,B 24.9493,C -1.6453,E1 24.9804,E2 186.7901} C_DIS
LIN {X -17.829,Y -104.8535,Z 109,A -103.9005,B 24.949,C -1.6495,E1 24.9725,E2 189.637} C_DIS
LIN {X -22.2788,Y -103.9993,Z 109,A -106.3528,B 24.949,C -1.65,E1 24.9658,E2 192.0909} C_DIS
LIN {X -25.1644,Y -103.3383,Z 109,A -108.0318,B 24.9491,C -1.6476,E1 24.9612,E2 193.778} C_DIS
LIN {X -30.5889,Y -101.8651,Z 109,A -110.7155,B 24.9482,C -1.663,E1 24.9541,E2 196.4293} C_DIS
LIN {X -34.1653,Y -100.7215,Z 109,A -113.1266,B 24.949,C -1.6494,E1 24.9476,E2 198.877} C_DIS
LIN {X -39.806,Y -98.6284,Z 109,A -116.2371,B 24.9485,C -1.6575,E1 24.9395,E2 201.9748} C_DIS
LIN {X -42.2746,Y -97.5959,Z 109,A -118.0987,B 24.9494,C -1.6429,E1 24.9346,E2 203.8755} C_DIS
LIN {X -46.3219,Y -95.7414,Z 109,A -120.2712,B 24.9487,C -1.6543,E1 24.9292,E2 206.0263} C_DIS
LIN {X -49.6099,Y -94.0792,Z 109,A -122.1615,B 24.9483,C -1.6605,E1 24.9245,E2 207.9071} C_DIS
LIN {X -52.5904,Y -92.4473,Z 109,A -124.0929,B 24.9484,C -1.6591,E1 24.9198,E2 209.8473} C_DIS
LIN {X -56.9284,Y -89.842,Z 109,A -126.6869,B 24.9479,C -1.6682,E1 24.9137,E2 212.4278} C_DIS
LIN {X -59.7587,Y -87.9828,Z 109,A -128.5433,B 24.9477,C -1.6699,E1 24.9093,E2 214.2862} C_DIS
LIN {X -63.0791,Y -85.6339,Z 109,A -130.659,B 24.9473,C -1.6765,E1 24.9045,E2 216.3936} C_DIS
LIN {X -65.3312,Y -83.9294,Z 109,A -133.2941,B 24.9497,C -1.6376,E1 24.8985,E2 219.1309} C_DIS
LIN {X -69.6716,Y -80.3621,Z 109,A -135.1293,B 24.9466,C -1.6878,E1 24.8949,E2 220.8538} C_DIS
LIN {X -72.15,Y -78.1431,Z 109,A -138.0772,B 24.9491,C -1.6485,E1 24.8886,E2 223.9071} C_DIS
LIN {X -76.0886,Y -74.3165,Z 109,A -140.0051,B 24.9463,C -1.6929,E1 24.885,E2 225.7376} C_DIS
LIN {X -80.1963,Y -69.8614,Z 109,A -143.2031,B 24.9457,C -1.7027,E1 24.879,E2 228.9264} C_DIS
LIN {X -81.8735,Y -67.888,Z 109,A -144.7834,B 24.9459,C -1.699,E1 24.8761,E2 230.5226} C_DIS
LIN {X -85.6526,Y -63.0535,Z 109,A -148.1457,B 24.9455,C -1.7049,E1 24.8704,E2 233.8868} C_DIS
LIN {X -87.7832,Y -60.0535,Z 109,A -150.2743,B 24.9455,C -1.7046,E1 24.8669,E2 236.0268} C_DIS
LIN {X -91.1628,Y -54.7864,Z 109,A -153.5199,B 24.9447,C -1.718,E1 24.8622,E2 239.2569} C_DIS
LIN {X -92.8739,Y -51.8313,Z 109,A -155.3265,B 24.9443,C -1.7242,E1 24.8597,E2 241.0581} C_DIS
LIN {X -94.248,Y -49.2894,Z 109,A -156.9733,B 24.9443,C -1.7252,E1 24.8575,E2 242.7114} C_DIS
LIN {X -95.8993,Y -45.9933,Z 109,A -158.9422,B 24.9438,C -1.7314,E1 24.8551,E2 244.6762} C_DIS
LIN {X -98.2256,Y -40.7932,Z 109,A -161.9723,B 24.9432,C -1.7416,E1 24.8517,E2 247.6986} C_DIS
LIN {X -99.4477,Y -37.712,Z 109,A -164.1705,B 24.9438,C -1.7319,E1 24.8494,E2 249.9322} C_DIS
LIN {X -101.1343,Y -32.9231,Z 109,A -166.509,B 24.9423,C -1.7544,E1 24.8474,E2 252.2303} C_DIS
LIN {X -102.0229,Y -30.0569,Z 109,A -168.1593,B 24.9421,C -1.7581,E1 24.846,E2 253.8814} C_DIS
LIN {X -102.9633,Y -26.6579,Z 109,A -170.0891,B 24.9418,C -1.7628,E1 24.8446,E2 255.8111} C_DIS
LIN {X -103.781,Y -23.2797,Z 109,A -172.1102,B 24.9418,C -1.7633,E1 24.8434,E2 257.8431} C_DIS
LIN {X -104.4917,Y -19.8394,Z 109,A -173.9971,B 24.9413,C -1.7694,E1 24.8423,E2 259.7265} C_DIS
LIN {X -105.1553,Y -15.9531,Z 109,A -176.3164,B 24.9413,C -1.7691,E1 24.8413,E2 262.0603} C_DIS
LIN {X -105.8125,Y -10.7638,Z 109,A -178.9284,B 24.9403,C -1.7855,E1 24.8405,E2 264.6489} C_DIS
LIN {X -106.1973,Y -5.8468,Z 109,A 178.1523,B 24.9403,C -1.7846,E1 24.8399,E2 267.5878} C_DIS
LIN {X -106.3549,Y -0.8952,Z 109,A 175.7499,B 24.9391,C -1.8027,E1 24.8398,E2 269.9614} C_DIS
LIN {X -106.3289,Y 2.5629,Z 109,A 173.6744,B 24.9391,C -1.8011,E1 24.8398,E2 272.0533} C_DIS
LIN {X -106.1373,Y 6.8565,Z 109,A 171.5435,B 24.9382,C -1.8153,E1 24.8402,E2 274.1633} C_DIS
LIN {X -105.8819,Y 10.057,Z 109,A 169.801,B 24.9379,C -1.8204,E1 24.8406,E2 275.904} C_DIS
LIN {X -105.4942,Y 13.5291,Z 109,A 167.9271,B 24.9374,C -1.8268,E1 24.8412,E2 277.7739} C_DIS
LIN {X -104.8688,Y 17.7375,Z 109,A 165.8759,B 24.9363,C -1.8428,E1 24.8421,E2 279.7991} C_DIS
LIN {X -104.4336,Y 20.1413,Z 109,A 164.294,B 24.9367,C -1.8375,E1 24.8429,E2 281.403} C_DIS
LIN {X -103.6674,Y 23.7726,Z 109,A 162.2829,B 24.9363,C -1.8435,E1 24.8441,E2 283.4117} C_DIS
LIN {X -102.5547,Y 28.1908,Z 109,A 159.6448,B 24.9363,C -1.8447,E1 24.846,E2 286.0622} C_DIS
LIN {X -101.4974,Y 31.7869,Z 109,A 157.8224,B 24.9353,C -1.8581,E1 24.8475,E2 287.8631} C_DIS
LIN {X -100.4134,Y 35.0603,Z 109,A 155.8765,B 24.9351,C -1.8607,E1 24.8492,E2 289.8139} C_DIS
LIN {X -99.0858,Y 38.6536,Z 109,A 153.8154,B 24.9346,C -1.8672,E1 24.8512,E2 291.8711} C_DIS
LIN {X -97.7708,Y 41.8724,Z 109,A 151.5704,B 24.9352,C -1.8596,E1 24.8537,E2 294.1468} C_DIS
LIN {X -95.653,Y 46.5059,Z 109,A 148.6059,B 24.9352,C -1.86,E1 24.8573,E2 297.1264} C_DIS
LIN {X -93.8625,Y 50.0214,Z 109,A 146.9622,B 24.9335,C -1.8835,E1 24.8594,E2 298.7228} C_DIS
LIN {X -90.1956,Y 56.3632,Z 109,A 143.4802,B 24.9315,C -1.9117,E1 24.8642,E2 302.1556} C_DIS
LIN {X -87.7034,Y 60.1713,Z 109,A 140.5461,B 24.9322,C -1.9011,E1 24.8688,E2 305.1298} C_DIS
LIN {X -84.0839,Y 65.1308,Z 109,A 137.8099,B 24.9301,C -1.9309,E1 24.8732,E2 307.8081} C_DIS
LIN {X -81.4702,Y 68.3734,Z 109,A 134.952,B 24.9313,C -1.9143,E1 24.8783,E2 310.7188} C_DIS
LIN {X -77.8643,Y 72.4519,Z 109,A 132.0691,B 24.9306,C -1.9236,E1 24.8837,E2 313.5926} C_DIS
LIN {X -76.1462,Y 74.2576,Z 109,A 130.6401,B 24.9306,C -1.9236,E1 24.8865,E2 315.0275} C_DIS
LIN {X -73.3678,Y 77.0038,Z 109,A 128.5071,B 24.9303,C -1.9277,E1 24.8907,E2 317.1598} C_DIS
LIN {X -68.0183,Y 81.7652,Z 109,A 124.7977,B 24.9293,C -1.9419,E1 24.8985,E2 320.8499} C_DIS
LIN {X -64.7177,Y 84.4022,Z 109,A 122.5697,B 24.9288,C -1.9486,E1 24.9034,E2 323.0703} C_DIS
LIN {X -62.5385,Y 86.0297,Z 109,A 120.6393,B 24.9298,C -1.9345,E1 24.9078,E2 325.0411} C_DIS
LIN {X -59.4045,Y 88.2226,Z 109,A 118.309,B 24.9303,C -1.9287,E1 24.9132,E2 327.393} C_DIS
LIN {X -56.0307,Y 90.4032,Z 109,A 116.4448,B 24.9292,C -1.9437,E1 24.9176,E2 329.2273} C_DIS
LIN {X -52.0963,Y 92.7259,Z 109,A 113.7181,B 24.9296,C -1.9383,E1 24.9242,E2 331.9749} C_DIS
LIN {X -48.7455,Y 94.5308,Z 109,A 112.3802,B 24.9274,C -1.9682,E1 24.9274,E2 333.2453} C_DIS
LIN {X -46.2227,Y 95.789,Z 109,A 110.6698,B 24.9277,C -1.9635,E1 24.9317,E2 334.9715} C_DIS
LIN {X -43.3036,Y 97.1444,Z 109,A 108.933,B 24.9275,C -1.966,E1 24.9361,E2 336.7066} C_DIS
LIN {X -40.2166,Y 98.4616,Z 109,A 106.372,B 24.9294,C -1.9404,E1 24.9429,E2 339.3341} C_DIS
LIN {X -35.8086,Y 100.1508,Z 109,A 104.6588,B 24.9269,C -1.9748,E1 24.9472,E2 340.9691} C_DIS
LIN {X -31.8948,Y 101.464,Z 109,A 102.1023,B 24.9276,C -1.9649,E1 24.954,E2 343.5538} C_DIS
LIN {X -27.1361,Y 102.8398,Z 109,A 99.559,B 24.9271,C -1.9724,E1 24.9609,E2 346.0833} C_DIS
LIN {X -23.656,Y 103.6944,Z 109,A 97.3332,B 24.9278,C -1.963,E1 24.967,E2 348.3343} C_DIS
LIN {X -20.4826,Y 104.3679,Z 109,A 96.0602,B 24.9263,C -1.9825,E1 24.9703,E2 349.5624} C_DIS
LIN {X -15.0463,Y 105.2885,Z 109,A 93.0347,B 24.9263,C -1.9825,E1 24.9787,E2 352.5907} C_DIS
LIN {X -11.8787,Y 105.6938,Z 109,A 90.6098,B 24.9282,C -1.9565,E1 24.9856,E2 355.0789} C_DIS
LIN {X -7.5765,Y 106.0887,Z 109,A 89.1522,B 24.9257,C -1.991,E1 24.9894,E2 356.4553} C_DIS
LIN {X -2.5322,Y 106.3294,Z 109,A 86.285,B 24.926,C -1.9861,E1 24.9975,E2 359.3347} C_DIS
LIN {X 4.1671,Y 106.2772,Z 109,A 82.8203,B 24.9256,C -1.9923,E1 25.0071,E2 362.7843} C_DIS
LIN {X 9.728,Y 105.9123,Z 109,A 79.9921,B 24.9251,C -1.999,E1 25.0149,E2 365.5953} C_DIS
LIN {X 14.861,Y 105.3148,Z 109,A 77.0336,B 24.9256,C -1.9916,E1 25.0232,E2 368.5692} C_DIS
LIN {X 18.9304,Y 104.6599,Z 109,A 74.6749,B 24.9261,C -1.9854,E1 25.0297,E2 370.9403} C_DIS
LIN {X 21.7978,Y 104.1013,Z 109,A 73.0115,B 24.9264,C -1.9811,E1 25.0343,E2 372.6118} C_DIS
LIN {X 27.5823,Y 102.7195,Z 109,A 70.1617,B 24.9255,C -1.9933,E1 25.0419,E2 375.4284} C_DIS
LIN {X 30.0716,Y 102.0185,Z 109,A 68.4404,B 24.9266,C -1.9792,E1 25.0466,E2 377.1803} C_DIS
LIN {X 33.1612,Y 101.0573,Z 109,A 66.242,B 24.928,C -1.9597,E1 25.0526,E2 379.4208} C_DIS
LIN {X 36.4407,Y 99.9206,Z 109,A 64.8736,B 24.9266,C -1.978,E1 25.056,E2 380.743} C_DIS
LIN {X 38.924,Y 98.9796,Z 109,A 63.4354,B 24.9268,C -1.9763,E1 25.0598,E2 382.1821} C_DIS
LIN {X 42.2215,Y 97.6191,Z 109,A 61.4993,B 24.927,C -1.9736,E1 25.0648,E2 384.12} C_DIS
LIN {X 45.0499,Y 96.3462,Z 109,A 59.7813,B 24.9273,C -1.9698,E1 25.0691,E2 385.8428} C_DIS
LIN {X 48.3351,Y 94.7405,Z 109,A 57.8981,B 24.9272,C -1.9708,E1 25.0738,E2 387.7184} C_DIS
LIN {X 50.9356,Y 93.3685,Z 109,A 55.8741,B 24.9286,C -1.9508,E1 25.0789,E2 389.7839} C_DIS
LIN {X 53.8293,Y 91.731,Z 109,A 54.4864,B 24.9276,C -1.9646,E1 25.0822,E2 391.1349} C_DIS
LIN {X 57.6738,Y 89.3636,Z 109,A 52.1751,B 24.9276,C -1.9658,E1 25.0876,E2 393.436} C_DIS
LIN {X 60.916,Y 87.1857,Z 109,A 49.9384,B 24.9282,C -1.9568,E1 25.0928,E2 395.6862} C_DIS
LIN {X 65.8673,Y 83.5078,Z 109,A 46.5336,B 24.9289,C -1.9475,E1 25.1004,E2 399.1008} C_DIS
LIN {X 68.4936,Y 81.37,Z 109,A 44.7093,B 24.9291,C -1.944,E1 25.1043,E2 400.9264} C_DIS
LIN {X 71.9762,Y 78.3038,Z 109,A 42.3642,B 24.9291,C -1.9454,E1 25.1092,E2 403.2589} C_DIS
LIN {X 74.6852,Y 75.7243,Z 109,A 40.3473,B 24.9294,C -1.9411,E1 25.1132,E2 405.2776} C_DIS
LIN {X 78.6434,Y 71.6052,Z 109,A 37.1937,B 24.9301,C -1.9311,E1 25.1193,E2 408.441} C_DIS
LIN {X 80.424,Y 69.6007,Z 109,A 35.7371,B 24.9304,C -1.9272,E1 25.122,E2 409.9001} C_DIS
LIN {X 82.6987,Y 66.8804,Z 109,A 34.0354,B 24.9301,C -1.9314,E1 25.125,E2 411.5841} C_DIS
LIN {X 84.676,Y 64.3614,Z 109,A 32.1491,B 24.9309,C -1.9204,E1 25.1282,E2 413.4874} C_DIS
LIN {X 87.6359,Y 60.2684,Z 109,A 29.6218,B 24.9308,C -1.9217,E1 25.1323,E2 415.9993} C_DIS
LIN {X 89.9837,Y 56.7023,Z 109,A 27.165,B 24.9317,C -1.9091,E1 25.136,E2 418.4735} C_DIS
LIN {X 91.9234,Y 53.5022,Z 109,A 25.1623,B 24.932,C -1.9043,E1 25.1389,E2 420.4775} C_DIS
LIN {X 93.5722,Y 50.56,Z 109,A 23.3781,B 24.9323,C -1.9007,E1 25.1413,E2 422.2607} C_DIS
LIN {X 95.9025,Y 45.9866,Z 109,A 20.0348,B 24.9345,C -1.8686,E1 25.1455,E2 425.6619} C_DIS
LIN {X 97.6981,Y 42.0391,Z 109,A 18.3394,B 24.9331,C -1.8889,E1 25.1473,E2 427.3003} C_DIS
LIN {X 99.1899,Y 38.3869,Z 109,A 16.1891,B 24.9336,C -1.8816,E1 25.1496,E2 429.4558} C_DIS
LIN {X 100.3537,Y 35.2305,Z 109,A 14.4739,B 24.9337,C -1.8803,E1 25.1512,E2 431.1643} C_DIS
LIN {X 101.433,Y 31.9947,Z 109,A 12.563,B 24.9343,C -1.8716,E1 25.1528,E2 433.0849} C_DIS
LIN {X 102.8992,Y 26.9071,Z 109,A 9.8569,B 24.9345,C -1.8691,E1 25.1549,E2 435.7814} C_DIS
LIN {X 103.6256,Y 23.9539,Z 109,A 8.1596,B 24.935,C -1.8615,E1 25.156,E2 437.4868} C_DIS
LIN {X 104.7722,Y 18.3057,Z 109,A 4.8053,B 24.9365,C -1.8411,E1 25.1578,E2 440.8697} C_DIS
LIN {X 105.6217,Y 12.4948,Z 109,A 1.9065,B 24.9364,C -1.8424,E1 25.1588,E2 443.7484} C_DIS
LIN {X 106.184,Y 6.0869,Z 109,A -2.2217,B 24.9391,C -1.803,E1 25.1597,E2 447.9449} C_DIS
LIN {X 106.349,Y 1.4714,Z 109,A -3.8458,B 24.9371,C -1.8318,E1 25.1597,E2 449.4914} C_DIS
LIN {X 106.2601,Y -4.5655,Z 109,A -7.1541,B 24.938,C -1.8189,E1 25.1597,E2 452.8106} C_DIS
LIN {X 106.043,Y -8.186,Z 109,A -8.8852,B 24.9378,C -1.8221,E1 25.1593,E2 454.5237} C_DIS
LIN {X 105.8092,Y -10.7951,Z 109,A -11.3011,B 24.941,C -1.7745,E1 25.1586,E2 457.0375} C_DIS
LIN {X 105.218,Y -15.5426,Z 109,A -13.0148,B 24.9391,C -1.803,E1 25.158,E2 458.6739} C_DIS
LIN {X 104.3672,Y -20.4863,Z 109,A -15.6714,B 24.9395,C -1.7963,E1 25.1567,E2 461.3309} C_DIS
LIN {X 103.8605,Y -22.9154,Z 109,A -17.2219,B 24.9404,C -1.7828,E1 25.1557,E2 462.9042} C_DIS
LIN {X 102.1337,Y -29.6833,Z 109,A -20.7413,B 24.9405,C -1.7812,E1 25.1532,E2 466.407} C_DIS
LIN {X 100.8969,Y -33.645,Z 109,A -24.4495,B 24.9451,C -1.7117,E1 25.1499,E2 470.2582} C_DIS
LIN {X 98.3668,Y -40.4494,Z 109,A -27.0593,B 24.9423,C -1.7546,E1 25.1473,E2 472.7523} C_DIS
LIN {X 95.261,Y -47.3011,Z 109,A -30.976,B 24.9427,C -1.7482,E1 25.1427,E2 476.6631} C_DIS
LIN {X 93.1918,Y -51.2613,Z 109,A -33.2866,B 24.9429,C -1.7451,E1 25.1397,E2 478.9688} C_DIS
LIN {X 91.1858,Y -54.748,Z 109,A -35.6136,B 24.9438,C -1.732,E1 25.1364,E2 481.3148} C_DIS
LIN {X 88.9641,Y -58.288,Z 109,A -37.8337,B 24.9441,C -1.7269,E1 25.133,E2 483.5357} C_DIS
LIN {X 87.1227,Y -61.0067,Z 109,A -39.4544,B 24.9441,C -1.7283,E1 25.1305,E2 485.1452} C_DIS
LIN {X 85.2109,Y -63.6492,Z 109,A -41.656,B 24.9455,C -1.7046,E1 25.1267,E2 487.3921} C_DIS
LIN {X 83.257,Y -66.1846,Z 109,A -43.6003,B 24.9464,C -1.6907,E1 25.1233,E2 489.3601} C_DIS
LIN {X 80.5826,Y -69.4178,Z 109,A -45.1408,B 24.9449,C -1.7152,E1 25.1206,E2 490.8358} C_DIS
LIN {X 78.6208,Y -71.6307,Z 109,A -47.5068,B 24.9472,C -1.6785,E1 25.1161,E2 493.2778} C_DIS
LIN {X 75.5823,Y -74.829,Z 109,A -49.808,B 24.9474,C -1.6758,E1 25.1115,E2 495.5755} C_DIS
LIN {X 72.5522,Y -77.7715,Z 109,A -51.3463,B 24.9458,C -1.7013,E1 25.1086,E2 497.0473} C_DIS
LIN {X 70.2612,Y -79.8472,Z 109,A -53.7606,B 24.948,C -1.6661,E1 25.1034,E2 499.5353} C_DIS
LIN {X 66.9937,Y -82.6069,Z 109,A -55.6784,B 24.9473,C -1.677,E1 25.0993,E2 501.4199} C_DIS
LIN {X 63.3404,Y -85.4426,Z 109,A -57.9972,B 24.9472,C -1.6789,E1 25.0941,E2 503.7259} C_DIS
LIN {X 58.7494,Y -88.6601,Z 109,A -60.946,B 24.9474,C -1.6758,E1 25.0874,E2 506.672} C_DIS
LIN {X 56.117,Y -90.3494,Z 109,A -62.4653,B 24.9471,C -1.6795,E1 25.0838,E2 508.1778} C_DIS
LIN {X 53.9436,Y -91.6634,Z 109,A -63.8295,B 24.9473,C -1.6771,E1 25.0805,E2 509.5434} C_DIS
LIN {X 51.3297,Y -93.154,Z 109,A -65.9067,B 24.9487,C -1.6552,E1 25.0754,E2 511.6661} C_DIS
LIN {X 44.9847,Y -96.3765,Z 109,A -69.8314,B 24.9493,C -1.6453,E1 25.0655,E2 515.6039} C_DIS
LIN {X 41.697,Y -97.8447,Z 109,A -71.2031,B 24.948,C -1.6657,E1 25.0621,E2 516.9239} C_DIS
LIN {X 35.7207,Y -100.1817,Z 109,A -74.6025,B 24.9482,C -1.6633,E1 25.0533,E2 520.3217} C_DIS
LIN {X 33.2362,Y -101.033,Z 109,A -76.24,B 24.9488,C -1.6524,E1 25.0488,E2 521.9818} C_DIS
LIN {X 28.4972,Y -102.4706,Z 109,A -78.9047,B 24.949,C -1.6495,E1 25.0417,E2 524.6489} C_DIS
LIN {X 24.8479,Y -103.4155,Z 109,A -80.7476,B 24.9487,C -1.6551,E1 25.0368,E2 526.4756} C_DIS
LIN {X 21.6628,Y -104.129,Z 109,A -83.5044,B 24.9512,C -1.6132,E1 25.029,E2 529.3281} C_DIS
LIN {X 16.4238,Y -105.0825,Z 109,A -85.1428,B 24.9483,C -1.6606,E1 25.0248,E2 530.8527} C_DIS
LIN {X 9.5793,Y -105.926,Z 109,A -88.9799,B 24.9488,C -1.6533,E1 25.0141,E2 534.7042} C_DIS
LIN {X 4.0007,Y -106.2843,Z 109,A -92.0696,B 24.9491,C -1.6488,E1 25.0055,E2 537.8033} C_DIS
LIN {X 0.7443,Y -106.332,Z 109,A -93.4219,B 24.9481,C -1.6649,E1 25.0018,E2 539.1173} C_DIS
Enddeposition()
LIN {X 0.7443,Y -106.332,Z 109,A -93.4219,B 24.9481,C -1.6649,E1 25.0018,E2 539.1173} C_DIS
Startdeposition()
$VEL.CP = VEL_PRINT
LIN {X 3.6089,Y -105.346,Z 109,A -91.6995,B 24.9466,C -1.6881,E1 25.0067,E2 537.3402} C_DIS
LIN {X 8.982,Y -105.0253,Z 109,A -88.5845,B 24.946,C -1.697,E1 25.0155,E2 534.2055} C_DIS
LIN {X 12.5427,Y -104.6586,Z 109,A -86.2507,B 24.9449,C -1.714,E1 25.0221,E2 531.833} C_DIS
LIN {X 16.0706,Y -104.1748,Z 109,A -84.7757,B 24.9461,C -1.6966,E1 25.026,E2 530.4008} C_DIS
LIN {X 21.0673,Y -103.2804,Z 109,A -82.0484,B 24.946,C -1.6975,E1 25.0335,E2 527.6743} C_DIS
LIN {X 24.666,Y -102.481,Z 109,A -80.0143,B 24.9458,C -1.7007,E1 25.039,E2 525.6355} C_DIS
LIN {X 27.6664,Y -101.7116,Z 109,A -77.8554,B 24.9444,C -1.7221,E1 25.045,E2 523.4294} C_DIS
LIN {X 31.2097,Y -100.6807,Z 109,A -76.3605,B 24.9456,C -1.7033,E1 25.0488,E2 521.9817} C_DIS
LIN {X 34.8372,Y -99.4838,Z 109,A -74.3033,B 24.9456,C -1.7051,E1 25.0543,E2 519.9242} C_DIS
LIN {X 39.6032,Y -97.6845,Z 109,A -71.5359,B 24.9453,C -1.7088,E1 25.0615,E2 517.154} C_DIS
LIN {X 42.8456,Y -96.3076,Z 109,A -69.5668,B 24.9449,C -1.714,E1 25.0666,E2 515.1776} C_DIS
LIN {X 48.5689,Y -93.5526,Z 109,A -66.0316,B 24.9444,C -1.723,E1 25.0755,E2 511.6304} C_DIS
LIN {X 52.0836,Y -91.6417,Z 109,A -63.9823,B 24.9444,C -1.7217,E1 25.0804,E2 509.5903} C_DIS
LIN {X 56.169,Y -89.1955,Z 109,A -61.7522,B 24.9451,C -1.7115,E1 25.0857,E2 507.3912} C_DIS
LIN {X 60.8745,Y -86.0531,Z 109,A -58.3834,B 24.9439,C -1.7299,E1 25.0936,E2 503.9903} C_DIS
LIN {X 63.4353,Y -84.1822,Z 109,A -56.6549,B 24.9437,C -1.7338,E1 25.0974,E2 502.2588} C_DIS
LIN {X 65.6224,Y -82.4892,Z 109,A -55.2337,B 24.9437,C -1.7336,E1 25.1005,E2 500.8434} C_DIS
LIN {X 68.7722,Y -79.8832,Z 109,A -52.8565,B 24.9429,C -1.7451,E1 25.1056,E2 498.4481} C_DIS
LIN {X 71.3747,Y -77.565,Z 109,A -51.0605,B 24.9429,C -1.7454,E1 25.1093,E2 496.6586} C_DIS
LIN {X 73.8203,Y -75.2419,Z 109,A -49.1201,B 24.9423,C -1.7544,E1 25.1133,E2 494.705} C_DIS
LIN {X 77.245,Y -71.7235,Z 109,A -46.4699,B 24.9419,C -1.7602,E1 25.1184,E2 492.0526} C_DIS
LIN {X 79.646,Y -69.0457,Z 109,A -44.5826,B 24.9418,C -1.7624,E1 25.1218,E2 490.1686} C_DIS
LIN {X 81.3255,Y -67.0595,Z 109,A -43.0879,B 24.9413,C -1.7696,E1 25.1245,E2 488.6638} C_DIS
LIN {X 84.0276,Y -63.6411,Z 109,A -40.8007,B 24.9411,C -1.7725,E1 25.1284,E2 486.3806} C_DIS
LIN {X 86.0626,Y -60.8612,Z 109,A -38.9198,B 24.9407,C -1.778,E1 25.1315,E2 484.4957} C_DIS
LIN {X 87.7263,Y -58.438,Z 109,A -37.1868,B 24.9401,C -1.7883,E1 25.1342,E2 482.747} C_DIS
LIN {X 89.4919,Y -55.6945,Z 109,A -34.8822,B 24.9382,C -1.8164,E1 25.1377,E2 480.3879} C_DIS
LIN {X 91.9522,Y -51.5313,Z 109,A -33.1818,B 24.9403,C -1.784,E1 25.1399,E2 478.7727} C_DIS
LIN {X 93.5042,Y -48.6609,Z 109,A -31.1764,B 24.9393,C -1.7992,E1 25.1426,E2 476.7421} C_DIS
LIN {X 95.7645,Y -44.046,Z 109,A -28.4841,B 24.9391,C -1.8033,E1 25.1458,E2 474.0547} C_DIS
LIN {X 97.0989,Y -41.0178,Z 109,A -26.7744,B 24.9389,C -1.8049,E1 25.1477,E2 472.3504} C_DIS
LIN {X 98.2928,Y -38.0713,Z 109,A -25.104,B 24.9387,C -1.8078,E1 25.1494,E2 470.6825} C_DIS
LIN {X 100.0924,Y -33.0541,Z 109,A -22.1743,B 24.938,C -1.8182,E1 25.1521,E2 467.7446} C_DIS
LIN {X 100.9721,Y -30.2551,Z 109,A -20.566,B 24.9376,C -1.8239,E1 25.1534,E2 466.1322} C_DIS
LIN {X 102.0935,Y -26.2217,Z 109,A -18.3241,B 24.9373,C -1.8297,E1 25.1551,E2 463.8895} C_DIS
LIN {X 102.8904,Y -22.9001,Z 109,A -16.3744,B 24.9366,C -1.8396,E1 25.1563,E2 461.9277} C_DIS
LIN {X 103.6259,Y -19.3061,Z 109,A -14.1761,B 24.9355,C -1.8549,E1 25.1575,E2 459.7063} C_DIS
LIN {X 104.4124,Y -14.4518,Z 109,A -11.5643,B 24.9351,C -1.8609,E1 25.1586,E2 457.0956} C_DIS
LIN {X 104.945,Y -9.8608,Z 109,A -9.3323,B 24.9354,C -1.8569,E1 25.1592,E2 454.8862} C_DIS
LIN {X 105.2174,Y -6.3419,Z 109,A -7.4592,B 24.9351,C -1.8611,E1 25.1596,E2 453.0142} C_DIS
LIN {X 105.3589,Y -3.1862,Z 109,A -5.1888,B 24.933,C -1.8907,E1 25.1598,E2 450.6876} C_DIS
LIN {X 105.4058,Y 0.5874,Z 109,A -3.66,B 24.9341,C -1.8747,E1 25.1598,E2 449.2057} C_DIS
LIN {X 105.229,Y 6.1325,Z 109,A -1.1414,B 24.9349,C -1.863,E1 25.1595,E2 446.7296} C_DIS
LIN {X 104.7574,Y 11.6987,Z 109,A 2.2128,B 24.9333,C -1.8863,E1 25.1587,E2 443.3404} C_DIS
LIN {X 103.9079,Y 17.7174,Z 109,A 5.6422,B 24.9322,C -1.9021,E1 25.1573,E2 439.8938} C_DIS
LIN {X 103.1202,Y 21.8464,Z 109,A 8.0213,B 24.9314,C -1.9133,E1 25.156,E2 437.5022} C_DIS
LIN {X 102.261,Y 25.5675,Z 109,A 10.1014,B 24.9309,C -1.9199,E1 25.1546,E2 435.4185} C_DIS
LIN {X 101.1426,Y 29.6804,Z 109,A 12.2201,B 24.9309,C -1.9185,E1 25.153,E2 433.3152} C_DIS
LIN {X 100.2494,Y 32.5689,Z 109,A 13.8917,B 24.9306,C -1.9247,E1 25.1516,E2 431.6387} C_DIS
LIN {X 99.0871,Y 35.9505,Z 109,A 15.5948,B 24.9309,C -1.9202,E1 25.15,E2 429.9557} C_DIS
LIN {X 97.7159,Y 39.5261,Z 109,A 17.8979,B 24.9297,C -1.9358,E1 25.1477,E2 427.6286} C_DIS
LIN {X 94.612,Y 46.469,Z 109,A 22.0813,B 24.9287,C -1.9496,E1 25.1428,E2 423.4352} C_DIS
LIN {X 92.8243,Y 49.9443,Z 109,A 24.1236,B 24.9286,C -1.952,E1 25.1401,E2 421.398} C_DIS
LIN {X 91.2437,Y 52.7762,Z 109,A 25.9134,B 24.9281,C -1.9579,E1 25.1377,E2 419.6035} C_DIS
LIN {X 89.5693,Y 55.5706,Z 109,A 27.3751,B 24.9287,C -1.9496,E1 25.1356,E2 418.1691} C_DIS
LIN {X 88.1641,Y 57.774,Z 109,A 29.0276,B 24.9277,C -1.9631,E1 25.133,E2 416.4931} C_DIS
LIN {X 86.3546,Y 60.4455,Z 109,A 30.9491,B 24.9269,C -1.9746,E1 25.13,E2 414.5536} C_DIS
LIN {X 83.9038,Y 63.8058,Z 109,A 33.1378,B 24.9267,C -1.9771,E1 25.1263,E2 412.3695} C_DIS
LIN {X 81.4116,Y 66.9558,Z 109,A 35.4774,B 24.9258,C -1.9889,E1 25.1222,E2 410.0129} C_DIS
LIN {X 78.9171,Y 69.8789,Z 109,A 38.3548,B 24.923,C -2.0271,E1 25.1167,E2 407.0582} C_DIS
LIN {X 74.8437,Y 74.2234,Z 109,A 40.5584,B 24.9257,C -1.9905,E1 25.1126,E2 404.9505} C_DIS
LIN {X 72.26,Y 76.7408,Z 109,A 42.3859,B 24.9258,C -1.989,E1 25.1089,E2 403.134} C_DIS
LIN {X 68.3038,Y 80.2823,Z 109,A 45.3192,B 24.9252,C -1.9967,E1 25.1028,E2 400.1942} C_DIS
LIN {X 61.8968,Y 85.3209,Z 109,A 49.8382,B 24.9244,C -2.0083,E1 25.0928,E2 395.6643} C_DIS
LIN {X 59.5156,Y 86.9989,Z 109,A 51.3847,B 24.9243,C -2.0094,E1 25.0892,E2 394.1205} C_DIS
LIN {X 56.3695,Y 89.0703,Z 109,A 53.6002,B 24.9235,C -2.0196,E1 25.084,E2 391.8882} C_DIS
LIN {X 52.8951,Y 91.1754,Z 109,A 55.6687,B 24.9237,C -2.0171,E1 25.079,E2 389.8319} C_DIS
LIN {X 49.3011,Y 93.1671,Z 109,A 57.7579,B 24.9239,C -2.0143,E1 25.0739,E2 387.7554} C_DIS
LIN {X 46.4076,Y 94.6424,Z 109,A 59.6486,B 24.9234,C -2.0216,E1 25.0692,E2 385.8524} C_DIS
LIN {X 43.2964,Y 96.1045,Z 109,A 61.4033,B 24.9236,C -2.0192,E1 25.0647,E2 384.1079} C_DIS
LIN {X 40.7786,Y 97.1997,Z 109,A 63.1686,B 24.9226,C -2.0319,E1 25.0601,E2 382.3167} C_DIS
LIN {X 37.1006,Y 98.6623,Z 109,A 65.6963,B 24.9213,C -2.0492,E1 25.0534,E2 379.7534} C_DIS
LIN {X 33.0185,Y 100.1039,Z 109,A 67.4946,B 24.9228,C -2.0287,E1 25.0488,E2 378.0072} C_DIS
LIN {X 29.3049,Y 101.2533,Z 109,A 69.5811,B 24.9228,C -2.0292,E1 25.0432,E2 375.9232} C_DIS
LIN {X 26.1481,Y 102.1124,Z 109,A 71.4401,B 24.9225,C -2.0335,E1 25.0382,E2 374.0568} C_DIS
LIN {X 21.8703,Y 103.115,Z 109,A 73.8292,B 24.9224,C -2.0348,E1 25.0317,E2 371.6679} C_DIS
LIN {X 17.9696,Y 103.8658,Z 109,A 76.0133,B 24.9222,C -2.0366,E1 25.0257,E2 369.482} C_DIS
LIN {X 13.2151,Y 104.5759,Z 109,A 78.7656,B 24.9218,C -2.0428,E1 25.018,E2 366.7173} C_DIS
LIN {X 8.4118,Y 105.0709,Z 109,A 81.0343,B 24.9228,C -2.0289,E1 25.0118,E2 364.4827} C_DIS
LIN {X 4.533,Y 105.3096,Z 109,A 83.2226,B 24.9226,C -2.0319,E1 25.0057,E2 362.2882} C_DIS
LIN {X -1.2603,Y 105.4013,Z 109,A 86.4578,B 24.9224,C -2.0346,E1 24.9966,E2 359.0468} C_DIS
LIN {X -5.1058,Y 105.2849,Z 109,A 88.3209,B 24.9231,C -2.0251,E1 24.9915,E2 357.206} C_DIS
LIN {X -9.1522,Y 105.0101,Z 109,A 90.8591,B 24.9222,C -2.0371,E1 24.9844,E2 354.6383} C_DIS
LIN {X -13.5439,Y 104.5333,Z 109,A 93.0307,B 24.923,C -2.0268,E1 24.9784,E2 352.4895} C_DIS
LIN {X -17.0226,Y 104.0241,Z 109,A 95.1317,B 24.9225,C -2.0328,E1 24.9726,E2 350.3725} C_DIS
LIN {X -20.8849,Y 103.3178,Z 109,A 97.1959,B 24.9229,C -2.0284,E1 24.9669,E2 348.3165} C_DIS
LIN {X -24.8008,Y 102.4481,Z 109,A 99.2529,B 24.9234,C -2.0216,E1 24.9614,E2 346.2727} C_DIS
LIN {X -28.2553,Y 101.5507,Z 109,A 101.1693,B 24.9236,C -2.0187,E1 24.9562,E2 344.3604} C_DIS
LIN {X -31.0496,Y 100.7304,Z 109,A 102.8821,B 24.9233,C -2.0219,E1 24.9516,E2 342.637} C_DIS
LIN {X -34.8342,Y 99.4849,Z 109,A 104.8046,B 24.9242,C -2.01,E1 24.9466,E2 340.7392} C_DIS
LIN {X -38.1776,Y 98.2511,Z 109,A 106.9249,B 24.9239,C -2.0144,E1 24.941,E2 338.6042} C_DIS
LIN {X -41.434,Y 96.9235,Z 109,A 108.9665,B 24.9237,C -2.0166,E1 24.9357,E2 336.5527} C_DIS
LIN {X -44.9556,Y 95.3411,Z 109,A 111.0639,B 24.924,C -2.0133,E1 24.9304,E2 334.4578} C_DIS
LIN {X -48.3246,Y 93.6779,Z 109,A 113.0586,B 24.9244,C -2.0082,E1 24.9255,E2 332.47} C_DIS
LIN {X -51.135,Y 92.1735,Z 109,A 114.7971,B 24.9246,C -2.0054,E1 24.9212,E2 330.7331} C_DIS
LIN {X -53.6925,Y 90.7071,Z 109,A 116.7643,B 24.9238,C -2.0162,E1 24.9164,E2 328.7342} C_DIS
LIN {X -56.6056,Y 88.9191,Z 109,A 118.6424,B 24.924,C -2.0134,E1 24.912,E2 326.8568} C_DIS
LIN {X -59.4757,Y 87.0259,Z 109,A 119.9957,B 24.9257,C -1.9905,E1 24.909,E2 325.5536} C_DIS
LIN {X -62.0849,Y 85.1831,Z 109,A 121.8094,B 24.9257,C -1.9898,E1 24.9048,E2 323.7352} C_DIS
LIN {X -64.4899,Y 83.3771,Z 109,A 123.6844,B 24.9254,C -1.9953,E1 24.9006,E2 321.8404} C_DIS
LIN {X -67.9246,Y 80.6053,Z 109,A 125.7464,B 24.9267,C -1.9775,E1 24.8963,E2 319.8129} C_DIS
LIN {X -71.52,Y 77.4316,Z 109,A 128.527,B 24.9267,C -1.9779,E1 24.8905,E2 317.0203} C_DIS
LIN {X -73.6004,Y 75.4587,Z 109,A 130.006,B 24.9271,C -1.9712,E1 24.8875,E2 315.551} C_DIS
LIN {X -76.351,Y 72.6745,Z 109,A 132.9683,B 24.9252,C -1.9968,E1 24.8816,E2 312.5149} C_DIS
LIN {X -79.4751,Y 69.2414,Z 109,A 134.7711,B 24.9277,C -1.9638,E1 24.8784,E2 310.7828} C_DIS
LIN {X -82.4116,Y 65.7206,Z 109,A 137.3003,B 24.9281,C -1.9586,E1 24.874,E2 308.2542} C_DIS
LIN {X -84.4972,Y 63.0159,Z 109,A 139.3637,B 24.9279,C -1.9611,E1 24.8705,E2 306.1748} C_DIS
LIN {X -86.9192,Y 59.6333,Z 109,A 141.4359,B 24.9289,C -1.9479,E1 24.8672,E2 304.1239} C_DIS
LIN {X -88.6104,Y 57.0865,Z 109,A 143.0059,B 24.9294,C -1.94,E1 24.8648,E2 302.565} C_DIS
LIN {X -91.5224,Y 52.2913,Z 109,A 146.1848,B 24.9297,C -1.9358,E1 24.8603,E2 299.3794} C_DIS
LIN {X -93.2726,Y 49.1006,Z 109,A 148.0846,B 24.9304,C -1.9272,E1 24.8577,E2 297.4902} C_DIS
LIN {X -94.6761,Y 46.3397,Z 109,A 150.2766,B 24.9294,C -1.9406,E1 24.855,E2 295.2544} C_DIS
LIN {X -96.1297,Y 43.2405,Z 109,A 151.7298,B 24.9309,C -1.9202,E1 24.8534,E2 293.842} C_DIS
LIN {X -97.559,Y 39.9115,Z 109,A 153.7218,B 24.9313,C -1.915,E1 24.8512,E2 291.8514} C_DIS
LIN {X -99.0197,Y 36.1352,Z 109,A 155.8532,B 24.9319,C -1.9057,E1 24.8491,E2 289.7302} C_DIS
LIN {X -100.3024,Y 32.4048,Z 109,A 157.9424,B 24.9325,C -1.897,E1 24.8473,E2 287.6498} C_DIS
LIN {X -102.2461,Y 25.6279,Z 109,A 161.943,B 24.933,C -1.8908,E1 24.8443,E2 283.6407} C_DIS
LIN {X -102.9728,Y 22.5226,Z 109,A 163.6763,B 24.9334,C -1.8853,E1 24.8432,E2 281.9103} C_DIS
LIN {X -103.7048,Y 18.8683,Z 109,A 165.5181,B 24.9343,C -1.8721,E1 24.8422,E2 280.089} C_DIS
LIN {X -104.1521,Y 16.2174,Z 109,A 167.2294,B 24.934,C -1.8764,E1 24.8415,E2 278.3573} C_DIS
LIN {X -104.6628,Y 12.5061,Z 109,A 169.221,B 24.9346,C -1.8682,E1 24.8408,E2 276.3734} C_DIS
LIN {X -104.9934,Y 9.3367,Z 109,A 170.8884,B 24.9351,C -1.8603,E1 24.8403,E2 274.7149} C_DIS
LIN {X -105.2265,Y 6.178,Z 109,A 172.6335,B 24.9355,C -1.8556,E1 24.84,E2 272.9706} C_DIS
LIN {X -105.3773,Y 2.5885,Z 109,A 174.664,B 24.9357,C -1.852,E1 24.8398,E2 270.9363} C_DIS
LIN {X -105.4051,Y -0.7098,Z 109,A 176.4637,B 24.9361,C -1.8465,E1 24.8398,E2 269.139} C_DIS
LIN {X -105.3199,Y -4.2929,Z 109,A 178.4644,B 24.9364,C -1.8421,E1 24.84,E2 267.1366} C_DIS
LIN {X -105.1039,Y -7.9993,Z 109,A -179.444,B 24.9367,C -1.8383,E1 24.8404,E2 265.0416} C_DIS
LIN {X -104.7373,Y -11.8702,Z 109,A -177.4684,B 24.9375,C -1.8265,E1 24.8409,E2 263.0822} C_DIS
LIN {X -104.4484,Y -14.1982,Z 109,A -176.0128,B 24.9373,C -1.829,E1 24.8415,E2 261.6119} C_DIS
LIN {X -103.8581,Y -18.0158,Z 109,A -173.9196,B 24.9378,C -1.8222,E1 24.8424,E2 259.5226} C_DIS
LIN {X -103.1287,Y -21.8063,Z 109,A -171.828,B 24.9382,C -1.8154,E1 24.8436,E2 257.435} C_DIS
LIN {X -102.3652,Y -25.1403,Z 109,A -170.0439,B 24.9388,C -1.8069,E1 24.8447,E2 255.6606} C_DIS
LIN {X -101.4332,Y -28.6699,Z 109,A -168.2576,B 24.9397,C -1.7936,E1 24.846,E2 253.8955} C_DIS
LIN {X -100.2371,Y -32.6068,Z 109,A -165.0865,B 24.9378,C -1.8211,E1 24.8488,E2 250.6407} C_DIS
LIN {X -98.758,Y -36.8481,Z 109,A -163.311,B 24.94,C -1.7893,E1 24.8504,E2 248.9309} C_DIS
LIN {X -97.5576,Y -39.9149,Z 109,A -161.5689,B 24.9405,C -1.7824,E1 24.8522,E2 247.1957} C_DIS
LIN {X -95.8237,Y -43.9187,Z 109,A -159.0646,B 24.9405,C -1.7804,E1 24.8551,E2 244.6823} C_DIS
LIN {X -94.33,Y -47.038,Z 109,A -157.1527,B 24.9409,C -1.7763,E1 24.8574,E2 242.7698} C_DIS
LIN {X -92.403,Y -50.7209,Z 109,A -154.7715,B 24.9409,C -1.7746,E1 24.8606,E2 240.3802} C_DIS
LIN {X -88.0983,Y -57.8738,Z 109,A -150.4055,B 24.9422,C -1.7562,E1 24.8669,E2 236.0356} C_DIS
LIN {X -86.0953,Y -60.8153,Z 109,A -148.431,B 24.9424,C -1.7528,E1 24.8701,E2 234.0595} C_DIS
LIN {X -84.5642,Y -62.9267,Z 109,A -146.836,B 24.9422,C -1.7559,E1 24.8728,E2 232.4494} C_DIS
LIN {X -81.8919,Y -66.3654,Z 109,A -144.6697,B 24.9431,C -1.7428,E1 24.8765,E2 230.3042} C_DIS
LIN {X -79.5767,Y -69.1251,Z 109,A -142.646,B 24.9432,C -1.7407,E1 24.8802,E2 228.2763} C_DIS
LIN {X -77.1123,Y -71.8649,Z 109,A -140.5996,B 24.9434,C -1.7378,E1 24.884,E2 226.2277} C_DIS
LIN {X -74.6055,Y -74.4646,Z 109,A -137.8045,B 24.9416,C -1.7651,E1 24.8897,E2 223.3558} C_DIS
LIN {X -70.7838,Y -78.107,Z 109,A -135.7014,B 24.9439,C -1.7301,E1 24.8939,E2 221.3273} C_DIS
LIN {X -67.9336,Y -80.5977,Z 109,A -133.8379,B 24.9446,C -1.7188,E1 24.8978,E2 219.4836} C_DIS
LIN {X -64.3567,Y -83.4798,Z 109,A -131.243,B 24.9446,C -1.718,E1 24.9035,E2 216.881} C_DIS
LIN {X -61.2209,Y -85.8059,Z 109,A -129.1379,B 24.945,C -1.7137,E1 24.9082,E2 214.7788} C_DIS
LIN {X -58.373,Y -87.7691,Z 109,A -127.1446,B 24.9449,C -1.7149,E1 24.9128,E2 212.7759} C_DIS
LIN {X -56.1712,Y -89.1941,Z 109,A -125.6972,B 24.9449,C -1.7135,E1 24.9163,E2 211.3271} C_DIS
LIN {X -53.1082,Y -91.0519,Z 109,A -123.8176,B 24.9453,C -1.7081,E1 24.9207,E2 209.4548} C_DIS
LIN {X -50.2095,Y -92.6804,Z 109,A -121.9858,B 24.9454,C -1.7066,E1 24.9252,E2 207.6213} C_DIS
LIN {X -46.9714,Y -94.363,Z 109,A -120.0475,B 24.9457,C -1.7023,E1 24.93,E2 205.6879} C_DIS
LIN {X -43.639,Y -95.9501,Z 109,A -117.8244,B 24.9453,C -1.7084,E1 24.9357,E2 203.4448} C_DIS
LIN {X -39.7116,Y -97.6404,Z 109,A -115.1258,B 24.9445,C -1.7207,E1 24.9428,E2 200.711} C_DIS
LIN {X -35.9974,Y -99.07,Z 109,A -113.5648,B 24.9462,C -1.6951,E1 24.9467,E2 199.2074} C_DIS
LIN {X -32.431,Y -100.294,Z 109,A -111.4828,B 24.9462,C -1.6947,E1 24.9522,E2 197.1225} C_DIS
LIN {X -29.2393,Y -101.2718,Z 109,A -109.4596,B 24.9457,C -1.7017,E1 24.9577,E2 195.0795} C_DIS
LIN {X -24.9215,Y -102.4186,Z 109,A -107.2335,B 24.9463,C -1.6923,E1 24.9637,E2 192.8724} C_DIS
LIN {X -21.1294,Y -103.2676,Z 109,A -105.0037,B 24.9461,C -1.696,E1 24.9698,E2 190.6311} C_DIS
LIN {X -17.3403,Y -103.971,Z 109,A -103.1935,B 24.9469,C -1.684,E1 24.9747,E2 188.8475} C_DIS
LIN {X -13.5114,Y -104.5375,Z 109,A -101.2783,B 24.9474,C -1.6761,E1 24.98,E2 186.9496} C_DIS
LIN {X -9.7037,Y -104.9593,Z 109,A -98.7245,B 24.9462,C -1.6945,E1 24.9872,E2 184.3505} C_DIS
LIN {X -5.0951,Y -105.2834,Z 109,A -95.9113,B 24.9454,C -1.7068,E1 24.9951,E2 181.5074} C_DIS
LIN {X -1.7403,Y -105.3929,Z 109,A -94.3323,B 24.946,C -1.6972,E1 24.9994,E2 179.951} C_DIS
LIN {X -1.7403,Y -105.3929,Z 109,A -94.3323,B 24.946,C -1.6972,E1 24.9994,E2 179.951} C_DIS
Enddeposition()
LIN {X 0.7171,Y -104.4509,Z 109,A -93.4729,B 24.9462,C -1.695,E1 25.0018,E2 179.0968} C_DIS
Startdeposition()
$VEL.CP = VEL_PRINT
LIN {X -1.8391,Y -104.4399,Z 109,A -95.4156,B 24.9475,C -1.6734,E1 24.9963,E2 181.0909} C_DIS
LIN {X -5.2548,Y -104.3251,Z 109,A -97.1889,B 24.9473,C -1.6771,E1 24.9913,E2 182.8556} C_DIS
LIN {X -8.303,Y -104.1255,Z 109,A -98.9136,B 24.9474,C -1.6752,E1 24.9865,E2 184.5855} C_DIS
LIN {X -11.5289,Y -103.8198,Z 109,A -100.8464,B 24.9478,C -1.6694,E1 24.9811,E2 186.5333} C_DIS
LIN {X -14.7935,Y -103.4032,Z 109,A -102.5491,B 24.9475,C -1.6737,E1 24.9764,E2 188.227} C_DIS
LIN {X -18.4102,Y -102.8209,Z 109,A -104.4781,B 24.9473,C -1.6774,E1 24.9711,E2 190.149} C_DIS
LIN {X -21.0969,Y -102.3035,Z 109,A -106.062,B 24.9474,C -1.6749,E1 24.9668,E2 191.7408} C_DIS
LIN {X -24.6787,Y -101.499,Z 109,A -107.992,B 24.9472,C -1.6791,E1 24.9615,E2 193.6633} C_DIS
LIN {X -27.1748,Y -100.8593,Z 109,A -109.4484,B 24.9472,C -1.6783,E1 24.9576,E2 195.1238} C_DIS
LIN {X -30.3294,Y -99.958,Z 109,A -111.4052,B 24.9475,C -1.6735,E1 24.9523,E2 197.0951} C_DIS
LIN {X -33.2994,Y -99.0062,Z 109,A -112.9644,B 24.9471,C -1.6807,E1 24.9482,E2 198.6402} C_DIS
LIN {X -36.4273,Y -97.9004,Z 109,A -114.9348,B 24.9473,C -1.6765,E1 24.943,E2 200.6244} C_DIS
LIN {X -39.315,Y -96.775,Z 109,A -116.4488,B 24.9468,C -1.6853,E1 24.9391,E2 202.121} C_DIS
LIN {X -41.8122,Y -95.7226,Z 109,A -118.0345,B 24.9469,C -1.6831,E1 24.935,E2 203.7155} C_DIS
LIN {X -45.174,Y -94.1827,Z 109,A -120.0148,B 24.9467,C -1.6873,E1 24.93,E2 205.6909} C_DIS
LIN {X -48.1102,Y -92.7194,Z 109,A -121.9735,B 24.9469,C -1.6835,E1 24.9251,E2 207.6637} C_DIS
LIN {X -50.9975,Y -91.161,Z 109,A -123.6694,B 24.9465,C -1.6899,E1 24.921,E2 209.3495} C_DIS
LIN {X -53.695,Y -89.6008,Z 109,A -125.4147,B 24.9465,C -1.691,E1 24.9168,E2 211.0973} C_DIS
LIN {X -56.3662,Y -87.9427,Z 109,A -127.0687,B 24.9461,C -1.6963,E1 24.9129,E2 212.744} C_DIS
LIN {X -59.0977,Y -86.1332,Z 109,A -128.8309,B 24.9458,C -1.7004,E1 24.9088,E2 214.5021} C_DIS
LIN {X -61.1953,Y -84.6558,Z 109,A -130.2443,B 24.9457,C -1.7026,E1 24.9056,E2 215.9154} C_DIS
LIN {X -63.6202,Y -82.8467,Z 109,A -131.9657,B 24.9457,C -1.7033,E1 24.9018,E2 217.6413} C_DIS
LIN {X -66.0005,Y -80.9635,Z 109,A -133.7376,B 24.9457,C -1.7024,E1 24.8979,E2 219.422} C_DIS
LIN {X -68.7144,Y -78.6727,Z 109,A -135.6087,B 24.9453,C -1.709,E1 24.8939,E2 221.2847} C_DIS
LIN {X -71.3832,Y -76.2599,Z 109,A -137.6079,B 24.9451,C -1.712,E1 24.8898,E2 223.2847} C_DIS
LIN {X -73.8891,Y -73.8365,Z 109,A -139.5721,B 24.9449,C -1.7141,E1 24.8859,E2 225.252} C_DIS
LIN {X -75.8367,Y -71.8332,Z 109,A -141.1016,B 24.9447,C -1.7176,E1 24.883,E2 226.7799} C_DIS
LIN {X -78.0213,Y -69.4538,Z 109,A -142.9174,B 24.9446,C -1.72,E1 24.8796,E2 228.5981} C_DIS
LIN {X -80.3386,Y -66.7591,Z 109,A -144.7921,B 24.9441,C -1.7273,E1 24.8762,E2 230.4642} C_DIS
LIN {X -82.564,Y -63.987,Z 109,A -146.7487,B 24.9438,C -1.7317,E1 24.8728,E2 232.4194} C_DIS
LIN {X -84.2334,Y -61.7722,Z 109,A -148.2109,B 24.9434,C -1.7376,E1 24.8704,E2 233.8746} C_DIS
LIN {X -85.9156,Y -59.4109,Z 109,A -149.9059,B 24.9434,C -1.7378,E1 24.8676,E2 235.5775} C_DIS
LIN {X -87.614,Y -56.8784,Z 109,A -151.6645,B 24.9434,C -1.739,E1 24.8649,E2 237.342} C_DIS
LIN {X -89.2404,Y -54.2883,Z 109,A -153.1742,B 24.9426,C -1.7495,E1 24.8627,E2 238.8345} C_DIS
LIN {X -90.5256,Y -52.1171,Z 109,A -154.5753,B 24.9424,C -1.7525,E1 24.8608,E2 240.2355} C_DIS
LIN {X -91.8604,Y -49.7268,Z 109,A -156.168,B 24.9424,C -1.7534,E1 24.8586,E2 241.8346} C_DIS
LIN {X -93.5522,Y -46.4658,Z 109,A -158.1514,B 24.9419,C -1.7601,E1 24.8561,E2 243.8126} C_DIS
LIN {X -94.9699,Y -43.4994,Z 109,A -160.1246,B 24.942,C -1.7591,E1 24.8538,E2 245.7988} C_DIS
LIN {X -96.3787,Y -40.278,Z 109,A -161.9012,B 24.9413,C -1.7701,E1 24.8518,E2 247.559} C_DIS
LIN {X -97.6558,Y -37.0731,Z 109,A -163.7814,B 24.9409,C -1.7761,E1 24.8499,E2 249.4355} C_DIS
LIN {X -98.5452,Y -34.6397,Z 109,A -165.2374,B 24.9407,C -1.7791,E1 24.8485,E2 250.8927} C_DIS
LIN {X -99.5783,Y -31.5536,Z 109,A -167.1972,B 24.9407,C -1.7782,E1 24.8468,E2 252.8657} C_DIS
LIN {X -100.476,Y -28.5595,Z 109,A -168.8004,B 24.9401,C -1.7874,E1 24.8456,E2 254.4562} C_DIS
LIN {X -101.3293,Y -25.374,Z 109,A -170.7392,B 24.9401,C -1.7884,E1 24.8442,E2 256.4042} C_DIS
LIN {X -102.0393,Y -22.3396,Z 109,A -172.2647,B 24.9393,C -1.8002,E1 24.8433,E2 257.9104} C_DIS
LIN {X -102.587,Y -19.6718,Z 109,A -173.8555,B 24.9392,C -1.8014,E1 24.8424,E2 259.5077} C_DIS
LIN {X -103.1317,Y -16.5933,Z 109,A -175.6957,B 24.9392,C -1.8024,E1 24.8416,E2 261.3564} C_DIS
LIN {X -103.6017,Y -13.3328,Z 109,A -177.4007,B 24.9385,C -1.8117,E1 24.841,E2 263.0494} C_DIS
LIN {X -104.0062,Y -9.6842,Z 109,A -179.3844,B 24.938,C -1.8192,E1 24.8404,E2 265.0271} C_DIS
LIN {X -104.2624,Y -6.3884,Z 109,A 178.6376,B 24.938,C -1.8192,E1 24.84,E2 267.017} C_DIS
LIN {X -104.4046,Y -3.2778,Z 109,A 177.07,B 24.9372,C -1.8297,E1 24.8398,E2 268.5691} C_DIS
LIN {X -104.4579,Y 0.0005,Z 109,A 175.1075,B 24.9372,C -1.8297,E1 24.8398,E2 270.5434} C_DIS
LIN {X -104.4046,Y 3.279,Z 109,A 173.3953,B 24.9366,C -1.8386,E1 24.8399,E2 272.2447} C_DIS
LIN {X -104.2609,Y 6.4134,Z 109,A 171.5599,B 24.9366,C -1.8401,E1 24.8402,E2 274.0875} C_DIS
LIN {X -104.0062,Y 9.6842,Z 109,A 169.8572,B 24.9359,C -1.8493,E1 24.8406,E2 275.7784} C_DIS
LIN {X -103.6014,Y 13.3355,Z 109,A 167.8716,B 24.9354,C -1.8569,E1 24.8412,E2 277.7579} C_DIS
Enddeposition()
END
